DECL E6POS XP241={X 672,Y -551,Z 95,A 0,B 0,C 180,S 6,T 16,E1 0.0,E2 0.0,E3 0.0,E4 0.0,E5 0.0,E6 0.0}
DECL FDAT FP241={TOOL_NO 4,BASE_NO 0,IPO_FRAME #BASE,POINT2[] " "}
DECL LDAT LCPDAT241={VEL 1,ACC 50.000,APO_DIST 500.000,APO_FAC 50.0000,AXIS_VEL 50.000,AXIS_ACC 50.000,ORI_TYP #VAR,CIRC_TYP #BASE,JERK_FAC 50.0000,GEAR_JERK 100.000,EXAX_IGN 0}

DECL E6POS XP242={X 672,Y -601,Z 95,A 0,B 0,C 180,S 6,T 16,E1 0.0,E2 0.0,E3 0.0,E4 0.0,E5 0.0,E6 0.0}
DECL FDAT FP242={TOOL_NO 4,BASE_NO 0,IPO_FRAME #BASE,POINT2[] " "}
DECL LDAT LCPDAT242={VEL 1,ACC 50.000,APO_DIST 500.000,APO_FAC 50.0000,AXIS_VEL 50.000,AXIS_ACC 50.000,ORI_TYP #VAR,CIRC_TYP #BASE,JERK_FAC 50.0000,GEAR_JERK 100.000,EXAX_IGN 0}

DECL E6POS XP243={X 672,Y -651,Z 95,A 0,B 0,C 180,S 6,T 16,E1 0.0,E2 0.0,E3 0.0,E4 0.0,E5 0.0,E6 0.0}
DECL FDAT FP243={TOOL_NO 4,BASE_NO 0,IPO_FRAME #BASE,POINT2[] " "}
DECL LDAT LCPDAT243={VEL 1,ACC 50.000,APO_DIST 500.000,APO_FAC 50.0000,AXIS_VEL 50.000,AXIS_ACC 50.000,ORI_TYP #VAR,CIRC_TYP #BASE,JERK_FAC 50.0000,GEAR_JERK 100.000,EXAX_IGN 0}

DECL E6POS XP244={X 672,Y -651,Z 145,A 0,B 0,C 180,S 6,T 16,E1 0.0,E2 0.0,E3 0.0,E4 0.0,E5 0.0,E6 0.0}
DECL FDAT FP244={TOOL_NO 4,BASE_NO 0,IPO_FRAME #BASE,POINT2[] " "}
DECL LDAT LCPDAT244={VEL 1,ACC 50.000,APO_DIST 500.000,APO_FAC 50.0000,AXIS_VEL 50.000,AXIS_ACC 50.000,ORI_TYP #VAR,CIRC_TYP #BASE,JERK_FAC 50.0000,GEAR_JERK 100.000,EXAX_IGN 0}

DECL E6POS XP245={X 672,Y -601,Z 145,A 0,B 0,C 180,S 6,T 16,E1 0.0,E2 0.0,E3 0.0,E4 0.0,E5 0.0,E6 0.0}
DECL FDAT FP245={TOOL_NO 4,BASE_NO 0,IPO_FRAME #BASE,POINT2[] " "}
DECL LDAT LCPDAT245={VEL 1,ACC 50.000,APO_DIST 500.000,APO_FAC 50.0000,AXIS_VEL 50.000,AXIS_ACC 50.000,ORI_TYP #VAR,CIRC_TYP #BASE,JERK_FAC 50.0000,GEAR_JERK 100.000,EXAX_IGN 0}

DECL E6POS XP246={X 672,Y -551,Z 145,A 0,B 0,C 180,S 6,T 16,E1 0.0,E2 0.0,E3 0.0,E4 0.0,E5 0.0,E6 0.0}
DECL FDAT FP246={TOOL_NO 4,BASE_NO 0,IPO_FRAME #BASE,POINT2[] " "}
DECL LDAT LCPDAT246={VEL 1,ACC 50.000,APO_DIST 500.000,APO_FAC 50.0000,AXIS_VEL 50.000,AXIS_ACC 50.000,ORI_TYP #VAR,CIRC_TYP #BASE,JERK_FAC 50.0000,GEAR_JERK 100.000,EXAX_IGN 0}

DECL E6POS XP247={X 672,Y -501,Z 145,A 0,B 0,C 180,S 6,T 16,E1 0.0,E2 0.0,E3 0.0,E4 0.0,E5 0.0,E6 0.0}
DECL FDAT FP247={TOOL_NO 4,BASE_NO 0,IPO_FRAME #BASE,POINT2[] " "}
DECL LDAT LCPDAT247={VEL 1,ACC 50.000,APO_DIST 500.000,APO_FAC 50.0000,AXIS_VEL 50.000,AXIS_ACC 50.000,ORI_TYP #VAR,CIRC_TYP #BASE,JERK_FAC 50.0000,GEAR_JERK 100.000,EXAX_IGN 0}

DECL E6POS XP248={X 672,Y -451,Z 145,A 0,B 0,C 180,S 6,T 16,E1 0.0,E2 0.0,E3 0.0,E4 0.0,E5 0.0,E6 0.0}
DECL FDAT FP248={TOOL_NO 4,BASE_NO 0,IPO_FRAME #BASE,POINT2[] " "}
DECL LDAT LCPDAT248={VEL 1,ACC 50.000,APO_DIST 500.000,APO_FAC 50.0000,AXIS_VEL 50.000,AXIS_ACC 50.000,ORI_TYP #VAR,CIRC_TYP #BASE,JERK_FAC 50.0000,GEAR_JERK 100.000,EXAX_IGN 0}

DECL E6POS XP249={X 672,Y -401,Z 145,A 0,B 0,C 180,S 6,T 16,E1 0.0,E2 0.0,E3 0.0,E4 0.0,E5 0.0,E6 0.0}
DECL FDAT FP249={TOOL_NO 4,BASE_NO 0,IPO_FRAME #BASE,POINT2[] " "}
DECL LDAT LCPDAT249={VEL 1,ACC 50.000,APO_DIST 500.000,APO_FAC 50.0000,AXIS_VEL 50.000,AXIS_ACC 50.000,ORI_TYP #VAR,CIRC_TYP #BASE,JERK_FAC 50.0000,GEAR_JERK 100.000,EXAX_IGN 0}

DECL E6POS XP250={X 672,Y -351,Z 145,A 0,B 0,C 180,S 6,T 16,E1 0.0,E2 0.0,E3 0.0,E4 0.0,E5 0.0,E6 0.0}
DECL FDAT FP250={TOOL_NO 4,BASE_NO 0,IPO_FRAME #BASE,POINT2[] " "}
DECL LDAT LCPDAT250={VEL 1,ACC 50.000,APO_DIST 500.000,APO_FAC 50.0000,AXIS_VEL 50.000,AXIS_ACC 50.000,ORI_TYP #VAR,CIRC_TYP #BASE,JERK_FAC 50.0000,GEAR_JERK 100.000,EXAX_IGN 0}

DECL E6POS XP251={X 672,Y -301,Z 145,A 0,B 0,C 180,S 6,T 16,E1 0.0,E2 0.0,E3 0.0,E4 0.0,E5 0.0,E6 0.0}
DECL FDAT FP251={TOOL_NO 4,BASE_NO 0,IPO_FRAME #BASE,POINT2[] " "}
DECL LDAT LCPDAT251={VEL 1,ACC 50.000,APO_DIST 500.000,APO_FAC 50.0000,AXIS_VEL 50.000,AXIS_ACC 50.000,ORI_TYP #VAR,CIRC_TYP #BASE,JERK_FAC 50.0000,GEAR_JERK 100.000,EXAX_IGN 0}

DECL E6POS XP252={X 672,Y -251,Z 145,A 0,B 0,C 180,S 6,T 16,E1 0.0,E2 0.0,E3 0.0,E4 0.0,E5 0.0,E6 0.0}
DECL FDAT FP252={TOOL_NO 4,BASE_NO 0,IPO_FRAME #BASE,POINT2[] " "}
DECL LDAT LCPDAT252={VEL 1,ACC 50.000,APO_DIST 500.000,APO_FAC 50.0000,AXIS_VEL 50.000,AXIS_ACC 50.000,ORI_TYP #VAR,CIRC_TYP #BASE,JERK_FAC 50.0000,GEAR_JERK 100.000,EXAX_IGN 0}

DECL E6POS XP253={X 672,Y -201,Z 145,A 0,B 0,C 180,S 6,T 16,E1 0.0,E2 0.0,E3 0.0,E4 0.0,E5 0.0,E6 0.0}
DECL FDAT FP253={TOOL_NO 4,BASE_NO 0,IPO_FRAME #BASE,POINT2[] " "}
DECL LDAT LCPDAT253={VEL 1,ACC 50.000,APO_DIST 500.000,APO_FAC 50.0000,AXIS_VEL 50.000,AXIS_ACC 50.000,ORI_TYP #VAR,CIRC_TYP #BASE,JERK_FAC 50.0000,GEAR_JERK 100.000,EXAX_IGN 0}

DECL E6POS XP254={X 672,Y -151,Z 145,A 0,B 0,C 180,S 6,T 16,E1 0.0,E2 0.0,E3 0.0,E4 0.0,E5 0.0,E6 0.0}
DECL FDAT FP254={TOOL_NO 4,BASE_NO 0,IPO_FRAME #BASE,POINT2[] " "}
DECL LDAT LCPDAT254={VEL 1,ACC 50.000,APO_DIST 500.000,APO_FAC 50.0000,AXIS_VEL 50.000,AXIS_ACC 50.000,ORI_TYP #VAR,CIRC_TYP #BASE,JERK_FAC 50.0000,GEAR_JERK 100.000,EXAX_IGN 0}

DECL E6POS XP255={X 672,Y -101,Z 145,A 0,B 0,C 180,S 6,T 16,E1 0.0,E2 0.0,E3 0.0,E4 0.0,E5 0.0,E6 0.0}
DECL FDAT FP255={TOOL_NO 4,BASE_NO 0,IPO_FRAME #BASE,POINT2[] " "}
DECL LDAT LCPDAT255={VEL 1,ACC 50.000,APO_DIST 500.000,APO_FAC 50.0000,AXIS_VEL 50.000,AXIS_ACC 50.000,ORI_TYP #VAR,CIRC_TYP #BASE,JERK_FAC 50.0000,GEAR_JERK 100.000,EXAX_IGN 0}

DECL E6POS XP256={X 672,Y -51,Z 145,A 0,B 0,C 180,S 6,T 16,E1 0.0,E2 0.0,E3 0.0,E4 0.0,E5 0.0,E6 0.0}
DECL FDAT FP256={TOOL_NO 4,BASE_NO 0,IPO_FRAME #BASE,POINT2[] " "}
DECL LDAT LCPDAT256={VEL 1,ACC 50.000,APO_DIST 500.000,APO_FAC 50.0000,AXIS_VEL 50.000,AXIS_ACC 50.000,ORI_TYP #VAR,CIRC_TYP #BASE,JERK_FAC 50.0000,GEAR_JERK 100.000,EXAX_IGN 0}

DECL E6POS XP257={X 672,Y -1,Z 145,A 0,B 0,C 180,S 6,T 16,E1 0.0,E2 0.0,E3 0.0,E4 0.0,E5 0.0,E6 0.0}
DECL FDAT FP257={TOOL_NO 4,BASE_NO 0,IPO_FRAME #BASE,POINT2[] " "}
DECL LDAT LCPDAT257={VEL 1,ACC 50.000,APO_DIST 500.000,APO_FAC 50.0000,AXIS_VEL 50.000,AXIS_ACC 50.000,ORI_TYP #VAR,CIRC_TYP #BASE,JERK_FAC 50.0000,GEAR_JERK 100.000,EXAX_IGN 0}

DECL E6POS XP258={X 672,Y 49,Z 145,A 0,B 0,C 180,S 6,T 16,E1 0.0,E2 0.0,E3 0.0,E4 0.0,E5 0.0,E6 0.0}
DECL FDAT FP258={TOOL_NO 4,BASE_NO 0,IPO_FRAME #BASE,POINT2[] " "}
DECL LDAT LCPDAT258={VEL 1,ACC 50.000,APO_DIST 500.000,APO_FAC 50.0000,AXIS_VEL 50.000,AXIS_ACC 50.000,ORI_TYP #VAR,CIRC_TYP #BASE,JERK_FAC 50.0000,GEAR_JERK 100.000,EXAX_IGN 0}

DECL E6POS XP259={X 672,Y 99,Z 145,A 0,B 0,C 180,S 6,T 16,E1 0.0,E2 0.0,E3 0.0,E4 0.0,E5 0.0,E6 0.0}
DECL FDAT FP259={TOOL_NO 4,BASE_NO 0,IPO_FRAME #BASE,POINT2[] " "}
DECL LDAT LCPDAT259={VEL 1,ACC 50.000,APO_DIST 500.000,APO_FAC 50.0000,AXIS_VEL 50.000,AXIS_ACC 50.000,ORI_TYP #VAR,CIRC_TYP #BASE,JERK_FAC 50.0000,GEAR_JERK 100.000,EXAX_IGN 0}

DECL E6POS XP260={X 672,Y 149,Z 145,A 0,B 0,C 180,S 6,T 16,E1 0.0,E2 0.0,E3 0.0,E4 0.0,E5 0.0,E6 0.0}
DECL FDAT FP260={TOOL_NO 4,BASE_NO 0,IPO_FRAME #BASE,POINT2[] " "}
DECL LDAT LCPDAT260={VEL 1,ACC 50.000,APO_DIST 500.000,APO_FAC 50.0000,AXIS_VEL 50.000,AXIS_ACC 50.000,ORI_TYP #VAR,CIRC_TYP #BASE,JERK_FAC 50.0000,GEAR_JERK 100.000,EXAX_IGN 0}

DECL E6POS XP261={X 672,Y 199,Z 145,A 0,B 0,C 180,S 6,T 16,E1 0.0,E2 0.0,E3 0.0,E4 0.0,E5 0.0,E6 0.0}
DECL FDAT FP261={TOOL_NO 4,BASE_NO 0,IPO_FRAME #BASE,POINT2[] " "}
DECL LDAT LCPDAT261={VEL 1,ACC 50.000,APO_DIST 500.000,APO_FAC 50.0000,AXIS_VEL 50.000,AXIS_ACC 50.000,ORI_TYP #VAR,CIRC_TYP #BASE,JERK_FAC 50.0000,GEAR_JERK 100.000,EXAX_IGN 0}

DECL E6POS XP262={X 672,Y 249,Z 145,A 0,B 0,C 180,S 6,T 16,E1 0.0,E2 0.0,E3 0.0,E4 0.0,E5 0.0,E6 0.0}
DECL FDAT FP262={TOOL_NO 4,BASE_NO 0,IPO_FRAME #BASE,POINT2[] " "}
DECL LDAT LCPDAT262={VEL 1,ACC 50.000,APO_DIST 500.000,APO_FAC 50.0000,AXIS_VEL 50.000,AXIS_ACC 50.000,ORI_TYP #VAR,CIRC_TYP #BASE,JERK_FAC 50.0000,GEAR_JERK 100.000,EXAX_IGN 0}

DECL E6POS XP263={X 672,Y 299,Z 145,A 0,B 0,C 180,S 6,T 16,E1 0.0,E2 0.0,E3 0.0,E4 0.0,E5 0.0,E6 0.0}
DECL FDAT FP263={TOOL_NO 4,BASE_NO 0,IPO_FRAME #BASE,POINT2[] " "}
DECL LDAT LCPDAT263={VEL 1,ACC 50.000,APO_DIST 500.000,APO_FAC 50.0000,AXIS_VEL 50.000,AXIS_ACC 50.000,ORI_TYP #VAR,CIRC_TYP #BASE,JERK_FAC 50.0000,GEAR_JERK 100.000,EXAX_IGN 0}

DECL E6POS XP264={X 672,Y 349,Z 145,A 0,B 0,C 180,S 6,T 16,E1 0.0,E2 0.0,E3 0.0,E4 0.0,E5 0.0,E6 0.0}
DECL FDAT FP264={TOOL_NO 4,BASE_NO 0,IPO_FRAME #BASE,POINT2[] " "}
DECL LDAT LCPDAT264={VEL 1,ACC 50.000,APO_DIST 500.000,APO_FAC 50.0000,AXIS_VEL 50.000,AXIS_ACC 50.000,ORI_TYP #VAR,CIRC_TYP #BASE,JERK_FAC 50.0000,GEAR_JERK 100.000,EXAX_IGN 0}

DECL E6POS XP265={X 672,Y 399,Z 145,A 0,B 0,C 180,S 6,T 16,E1 0.0,E2 0.0,E3 0.0,E4 0.0,E5 0.0,E6 0.0}
DECL FDAT FP265={TOOL_NO 4,BASE_NO 0,IPO_FRAME #BASE,POINT2[] " "}
DECL LDAT LCPDAT265={VEL 1,ACC 50.000,APO_DIST 500.000,APO_FAC 50.0000,AXIS_VEL 50.000,AXIS_ACC 50.000,ORI_TYP #VAR,CIRC_TYP #BASE,JERK_FAC 50.0000,GEAR_JERK 100.000,EXAX_IGN 0}

DECL E6POS XP266={X 672,Y 449,Z 145,A 0,B 0,C 180,S 6,T 16,E1 0.0,E2 0.0,E3 0.0,E4 0.0,E5 0.0,E6 0.0}
DECL FDAT FP266={TOOL_NO 4,BASE_NO 0,IPO_FRAME #BASE,POINT2[] " "}
DECL LDAT LCPDAT266={VEL 1,ACC 50.000,APO_DIST 500.000,APO_FAC 50.0000,AXIS_VEL 50.000,AXIS_ACC 50.000,ORI_TYP #VAR,CIRC_TYP #BASE,JERK_FAC 50.0000,GEAR_JERK 100.000,EXAX_IGN 0}

DECL E6POS XP267={X 672,Y 499,Z 145,A 0,B 0,C 180,S 6,T 16,E1 0.0,E2 0.0,E3 0.0,E4 0.0,E5 0.0,E6 0.0}
DECL FDAT FP267={TOOL_NO 4,BASE_NO 0,IPO_FRAME #BASE,POINT2[] " "}
DECL LDAT LCPDAT267={VEL 1,ACC 50.000,APO_DIST 500.000,APO_FAC 50.0000,AXIS_VEL 50.000,AXIS_ACC 50.000,ORI_TYP #VAR,CIRC_TYP #BASE,JERK_FAC 50.0000,GEAR_JERK 100.000,EXAX_IGN 0}

DECL E6POS XP268={X 672,Y 499,Z 195,A 0,B 0,C 180,S 6,T 16,E1 0.0,E2 0.0,E3 0.0,E4 0.0,E5 0.0,E6 0.0}
DECL FDAT FP268={TOOL_NO 4,BASE_NO 0,IPO_FRAME #BASE,POINT2[] " "}
DECL LDAT LCPDAT268={VEL 1,ACC 50.000,APO_DIST 500.000,APO_FAC 50.0000,AXIS_VEL 50.000,AXIS_ACC 50.000,ORI_TYP #VAR,CIRC_TYP #BASE,JERK_FAC 50.0000,GEAR_JERK 100.000,EXAX_IGN 0}

DECL E6POS XP269={X 672,Y 449,Z 195,A 0,B 0,C 180,S 6,T 16,E1 0.0,E2 0.0,E3 0.0,E4 0.0,E5 0.0,E6 0.0}
DECL FDAT FP269={TOOL_NO 4,BASE_NO 0,IPO_FRAME #BASE,POINT2[] " "}
DECL LDAT LCPDAT269={VEL 1,ACC 50.000,APO_DIST 500.000,APO_FAC 50.0000,AXIS_VEL 50.000,AXIS_ACC 50.000,ORI_TYP #VAR,CIRC_TYP #BASE,JERK_FAC 50.0000,GEAR_JERK 100.000,EXAX_IGN 0}

DECL E6POS XP270={X 672,Y 399,Z 195,A 0,B 0,C 180,S 6,T 16,E1 0.0,E2 0.0,E3 0.0,E4 0.0,E5 0.0,E6 0.0}
DECL FDAT FP270={TOOL_NO 4,BASE_NO 0,IPO_FRAME #BASE,POINT2[] " "}
DECL LDAT LCPDAT270={VEL 1,ACC 50.000,APO_DIST 500.000,APO_FAC 50.0000,AXIS_VEL 50.000,AXIS_ACC 50.000,ORI_TYP #VAR,CIRC_TYP #BASE,JERK_FAC 50.0000,GEAR_JERK 100.000,EXAX_IGN 0}

DECL E6POS XP271={X 672,Y 349,Z 195,A 0,B 0,C 180,S 6,T 16,E1 0.0,E2 0.0,E3 0.0,E4 0.0,E5 0.0,E6 0.0}
DECL FDAT FP271={TOOL_NO 4,BASE_NO 0,IPO_FRAME #BASE,POINT2[] " "}
DECL LDAT LCPDAT271={VEL 1,ACC 50.000,APO_DIST 500.000,APO_FAC 50.0000,AXIS_VEL 50.000,AXIS_ACC 50.000,ORI_TYP #VAR,CIRC_TYP #BASE,JERK_FAC 50.0000,GEAR_JERK 100.000,EXAX_IGN 0}

DECL E6POS XP272={X 672,Y 299,Z 195,A 0,B 0,C 180,S 6,T 16,E1 0.0,E2 0.0,E3 0.0,E4 0.0,E5 0.0,E6 0.0}
DECL FDAT FP272={TOOL_NO 4,BASE_NO 0,IPO_FRAME #BASE,POINT2[] " "}
DECL LDAT LCPDAT272={VEL 1,ACC 50.000,APO_DIST 500.000,APO_FAC 50.0000,AXIS_VEL 50.000,AXIS_ACC 50.000,ORI_TYP #VAR,CIRC_TYP #BASE,JERK_FAC 50.0000,GEAR_JERK 100.000,EXAX_IGN 0}

DECL E6POS XP273={X 672,Y 249,Z 195,A 0,B 0,C 180,S 6,T 16,E1 0.0,E2 0.0,E3 0.0,E4 0.0,E5 0.0,E6 0.0}
DECL FDAT FP273={TOOL_NO 4,BASE_NO 0,IPO_FRAME #BASE,POINT2[] " "}
DECL LDAT LCPDAT273={VEL 1,ACC 50.000,APO_DIST 500.000,APO_FAC 50.0000,AXIS_VEL 50.000,AXIS_ACC 50.000,ORI_TYP #VAR,CIRC_TYP #BASE,JERK_FAC 50.0000,GEAR_JERK 100.000,EXAX_IGN 0}

DECL E6POS XP274={X 672,Y 199,Z 195,A 0,B 0,C 180,S 6,T 16,E1 0.0,E2 0.0,E3 0.0,E4 0.0,E5 0.0,E6 0.0}
DECL FDAT FP274={TOOL_NO 4,BASE_NO 0,IPO_FRAME #BASE,POINT2[] " "}
DECL LDAT LCPDAT274={VEL 1,ACC 50.000,APO_DIST 500.000,APO_FAC 50.0000,AXIS_VEL 50.000,AXIS_ACC 50.000,ORI_TYP #VAR,CIRC_TYP #BASE,JERK_FAC 50.0000,GEAR_JERK 100.000,EXAX_IGN 0}

DECL E6POS XP275={X 672,Y 149,Z 195,A 0,B 0,C 180,S 6,T 16,E1 0.0,E2 0.0,E3 0.0,E4 0.0,E5 0.0,E6 0.0}
DECL FDAT FP275={TOOL_NO 4,BASE_NO 0,IPO_FRAME #BASE,POINT2[] " "}
DECL LDAT LCPDAT275={VEL 1,ACC 50.000,APO_DIST 500.000,APO_FAC 50.0000,AXIS_VEL 50.000,AXIS_ACC 50.000,ORI_TYP #VAR,CIRC_TYP #BASE,JERK_FAC 50.0000,GEAR_JERK 100.000,EXAX_IGN 0}

DECL E6POS XP276={X 672,Y 99,Z 195,A 0,B 0,C 180,S 6,T 16,E1 0.0,E2 0.0,E3 0.0,E4 0.0,E5 0.0,E6 0.0}
DECL FDAT FP276={TOOL_NO 4,BASE_NO 0,IPO_FRAME #BASE,POINT2[] " "}
DECL LDAT LCPDAT276={VEL 1,ACC 50.000,APO_DIST 500.000,APO_FAC 50.0000,AXIS_VEL 50.000,AXIS_ACC 50.000,ORI_TYP #VAR,CIRC_TYP #BASE,JERK_FAC 50.0000,GEAR_JERK 100.000,EXAX_IGN 0}

DECL E6POS XP277={X 672,Y 49,Z 195,A 0,B 0,C 180,S 6,T 16,E1 0.0,E2 0.0,E3 0.0,E4 0.0,E5 0.0,E6 0.0}
DECL FDAT FP277={TOOL_NO 4,BASE_NO 0,IPO_FRAME #BASE,POINT2[] " "}
DECL LDAT LCPDAT277={VEL 1,ACC 50.000,APO_DIST 500.000,APO_FAC 50.0000,AXIS_VEL 50.000,AXIS_ACC 50.000,ORI_TYP #VAR,CIRC_TYP #BASE,JERK_FAC 50.0000,GEAR_JERK 100.000,EXAX_IGN 0}

DECL E6POS XP278={X 672,Y -1,Z 195,A 0,B 0,C 180,S 6,T 16,E1 0.0,E2 0.0,E3 0.0,E4 0.0,E5 0.0,E6 0.0}
DECL FDAT FP278={TOOL_NO 4,BASE_NO 0,IPO_FRAME #BASE,POINT2[] " "}
DECL LDAT LCPDAT278={VEL 1,ACC 50.000,APO_DIST 500.000,APO_FAC 50.0000,AXIS_VEL 50.000,AXIS_ACC 50.000,ORI_TYP #VAR,CIRC_TYP #BASE,JERK_FAC 50.0000,GEAR_JERK 100.000,EXAX_IGN 0}

DECL E6POS XP279={X 672,Y -51,Z 195,A 0,B 0,C 180,S 6,T 16,E1 0.0,E2 0.0,E3 0.0,E4 0.0,E5 0.0,E6 0.0}
DECL FDAT FP279={TOOL_NO 4,BASE_NO 0,IPO_FRAME #BASE,POINT2[] " "}
DECL LDAT LCPDAT279={VEL 1,ACC 50.000,APO_DIST 500.000,APO_FAC 50.0000,AXIS_VEL 50.000,AXIS_ACC 50.000,ORI_TYP #VAR,CIRC_TYP #BASE,JERK_FAC 50.0000,GEAR_JERK 100.000,EXAX_IGN 0}

DECL E6POS XP280={X 672,Y -101,Z 195,A 0,B 0,C 180,S 6,T 16,E1 0.0,E2 0.0,E3 0.0,E4 0.0,E5 0.0,E6 0.0}
DECL FDAT FP280={TOOL_NO 4,BASE_NO 0,IPO_FRAME #BASE,POINT2[] " "}
DECL LDAT LCPDAT280={VEL 1,ACC 50.000,APO_DIST 500.000,APO_FAC 50.0000,AXIS_VEL 50.000,AXIS_ACC 50.000,ORI_TYP #VAR,CIRC_TYP #BASE,JERK_FAC 50.0000,GEAR_JERK 100.000,EXAX_IGN 0}

DECL E6POS XP281={X 672,Y -151,Z 195,A 0,B 0,C 180,S 6,T 16,E1 0.0,E2 0.0,E3 0.0,E4 0.0,E5 0.0,E6 0.0}
DECL FDAT FP281={TOOL_NO 4,BASE_NO 0,IPO_FRAME #BASE,POINT2[] " "}
DECL LDAT LCPDAT281={VEL 1,ACC 50.000,APO_DIST 500.000,APO_FAC 50.0000,AXIS_VEL 50.000,AXIS_ACC 50.000,ORI_TYP #VAR,CIRC_TYP #BASE,JERK_FAC 50.0000,GEAR_JERK 100.000,EXAX_IGN 0}

DECL E6POS XP282={X 672,Y -201,Z 195,A 0,B 0,C 180,S 6,T 16,E1 0.0,E2 0.0,E3 0.0,E4 0.0,E5 0.0,E6 0.0}
DECL FDAT FP282={TOOL_NO 4,BASE_NO 0,IPO_FRAME #BASE,POINT2[] " "}
DECL LDAT LCPDAT282={VEL 1,ACC 50.000,APO_DIST 500.000,APO_FAC 50.0000,AXIS_VEL 50.000,AXIS_ACC 50.000,ORI_TYP #VAR,CIRC_TYP #BASE,JERK_FAC 50.0000,GEAR_JERK 100.000,EXAX_IGN 0}

DECL E6POS XP283={X 672,Y -251,Z 195,A 0,B 0,C 180,S 6,T 16,E1 0.0,E2 0.0,E3 0.0,E4 0.0,E5 0.0,E6 0.0}
DECL FDAT FP283={TOOL_NO 4,BASE_NO 0,IPO_FRAME #BASE,POINT2[] " "}
DECL LDAT LCPDAT283={VEL 1,ACC 50.000,APO_DIST 500.000,APO_FAC 50.0000,AXIS_VEL 50.000,AXIS_ACC 50.000,ORI_TYP #VAR,CIRC_TYP #BASE,JERK_FAC 50.0000,GEAR_JERK 100.000,EXAX_IGN 0}

DECL E6POS XP284={X 672,Y -301,Z 195,A 0,B 0,C 180,S 6,T 16,E1 0.0,E2 0.0,E3 0.0,E4 0.0,E5 0.0,E6 0.0}
DECL FDAT FP284={TOOL_NO 4,BASE_NO 0,IPO_FRAME #BASE,POINT2[] " "}
DECL LDAT LCPDAT284={VEL 1,ACC 50.000,APO_DIST 500.000,APO_FAC 50.0000,AXIS_VEL 50.000,AXIS_ACC 50.000,ORI_TYP #VAR,CIRC_TYP #BASE,JERK_FAC 50.0000,GEAR_JERK 100.000,EXAX_IGN 0}

DECL E6POS XP285={X 672,Y -351,Z 195,A 0,B 0,C 180,S 6,T 16,E1 0.0,E2 0.0,E3 0.0,E4 0.0,E5 0.0,E6 0.0}
DECL FDAT FP285={TOOL_NO 4,BASE_NO 0,IPO_FRAME #BASE,POINT2[] " "}
DECL LDAT LCPDAT285={VEL 1,ACC 50.000,APO_DIST 500.000,APO_FAC 50.0000,AXIS_VEL 50.000,AXIS_ACC 50.000,ORI_TYP #VAR,CIRC_TYP #BASE,JERK_FAC 50.0000,GEAR_JERK 100.000,EXAX_IGN 0}

DECL E6POS XP286={X 672,Y -401,Z 195,A 0,B 0,C 180,S 6,T 16,E1 0.0,E2 0.0,E3 0.0,E4 0.0,E5 0.0,E6 0.0}
DECL FDAT FP286={TOOL_NO 4,BASE_NO 0,IPO_FRAME #BASE,POINT2[] " "}
DECL LDAT LCPDAT286={VEL 1,ACC 50.000,APO_DIST 500.000,APO_FAC 50.0000,AXIS_VEL 50.000,AXIS_ACC 50.000,ORI_TYP #VAR,CIRC_TYP #BASE,JERK_FAC 50.0000,GEAR_JERK 100.000,EXAX_IGN 0}

DECL E6POS XP287={X 672,Y -451,Z 195,A 0,B 0,C 180,S 6,T 16,E1 0.0,E2 0.0,E3 0.0,E4 0.0,E5 0.0,E6 0.0}
DECL FDAT FP287={TOOL_NO 4,BASE_NO 0,IPO_FRAME #BASE,POINT2[] " "}
DECL LDAT LCPDAT287={VEL 1,ACC 50.000,APO_DIST 500.000,APO_FAC 50.0000,AXIS_VEL 50.000,AXIS_ACC 50.000,ORI_TYP #VAR,CIRC_TYP #BASE,JERK_FAC 50.0000,GEAR_JERK 100.000,EXAX_IGN 0}

DECL E6POS XP288={X 672,Y -501,Z 195,A 0,B 0,C 180,S 6,T 16,E1 0.0,E2 0.0,E3 0.0,E4 0.0,E5 0.0,E6 0.0}
DECL FDAT FP288={TOOL_NO 4,BASE_NO 0,IPO_FRAME #BASE,POINT2[] " "}
DECL LDAT LCPDAT288={VEL 1,ACC 50.000,APO_DIST 500.000,APO_FAC 50.0000,AXIS_VEL 50.000,AXIS_ACC 50.000,ORI_TYP #VAR,CIRC_TYP #BASE,JERK_FAC 50.0000,GEAR_JERK 100.000,EXAX_IGN 0}

DECL E6POS XP289={X 672,Y -551,Z 195,A 0,B 0,C 180,S 6,T 16,E1 0.0,E2 0.0,E3 0.0,E4 0.0,E5 0.0,E6 0.0}
DECL FDAT FP289={TOOL_NO 4,BASE_NO 0,IPO_FRAME #BASE,POINT2[] " "}
DECL LDAT LCPDAT289={VEL 1,ACC 50.000,APO_DIST 500.000,APO_FAC 50.0000,AXIS_VEL 50.000,AXIS_ACC 50.000,ORI_TYP #VAR,CIRC_TYP #BASE,JERK_FAC 50.0000,GEAR_JERK 100.000,EXAX_IGN 0}

DECL E6POS XP290={X 672,Y -601,Z 195,A 0,B 0,C 180,S 6,T 16,E1 0.0,E2 0.0,E3 0.0,E4 0.0,E5 0.0,E6 0.0}
DECL FDAT FP290={TOOL_NO 4,BASE_NO 0,IPO_FRAME #BASE,POINT2[] " "}
DECL LDAT LCPDAT290={VEL 1,ACC 50.000,APO_DIST 500.000,APO_FAC 50.0000,AXIS_VEL 50.000,AXIS_ACC 50.000,ORI_TYP #VAR,CIRC_TYP #BASE,JERK_FAC 50.0000,GEAR_JERK 100.000,EXAX_IGN 0}

DECL E6POS XP291={X 672,Y -651,Z 195,A 0,B 0,C 180,S 6,T 16,E1 0.0,E2 0.0,E3 0.0,E4 0.0,E5 0.0,E6 0.0}
DECL FDAT FP291={TOOL_NO 4,BASE_NO 0,IPO_FRAME #BASE,POINT2[] " "}
DECL LDAT LCPDAT291={VEL 1,ACC 50.000,APO_DIST 500.000,APO_FAC 50.0000,AXIS_VEL 50.000,AXIS_ACC 50.000,ORI_TYP #VAR,CIRC_TYP #BASE,JERK_FAC 50.0000,GEAR_JERK 100.000,EXAX_IGN 0}

DECL E6POS XP292={X 672,Y -651,Z 245,A 0,B 0,C 180,S 6,T 16,E1 0.0,E2 0.0,E3 0.0,E4 0.0,E5 0.0,E6 0.0}
DECL FDAT FP292={TOOL_NO 4,BASE_NO 0,IPO_FRAME #BASE,POINT2[] " "}
DECL LDAT LCPDAT292={VEL 1,ACC 50.000,APO_DIST 500.000,APO_FAC 50.0000,AXIS_VEL 50.000,AXIS_ACC 50.000,ORI_TYP #VAR,CIRC_TYP #BASE,JERK_FAC 50.0000,GEAR_JERK 100.000,EXAX_IGN 0}

DECL E6POS XP293={X 672,Y -601,Z 245,A 0,B 0,C 180,S 6,T 16,E1 0.0,E2 0.0,E3 0.0,E4 0.0,E5 0.0,E6 0.0}
DECL FDAT FP293={TOOL_NO 4,BASE_NO 0,IPO_FRAME #BASE,POINT2[] " "}
DECL LDAT LCPDAT293={VEL 1,ACC 50.000,APO_DIST 500.000,APO_FAC 50.0000,AXIS_VEL 50.000,AXIS_ACC 50.000,ORI_TYP #VAR,CIRC_TYP #BASE,JERK_FAC 50.0000,GEAR_JERK 100.000,EXAX_IGN 0}

DECL E6POS XP294={X 672,Y -551,Z 245,A 0,B 0,C 180,S 6,T 16,E1 0.0,E2 0.0,E3 0.0,E4 0.0,E5 0.0,E6 0.0}
DECL FDAT FP294={TOOL_NO 4,BASE_NO 0,IPO_FRAME #BASE,POINT2[] " "}
DECL LDAT LCPDAT294={VEL 1,ACC 50.000,APO_DIST 500.000,APO_FAC 50.0000,AXIS_VEL 50.000,AXIS_ACC 50.000,ORI_TYP #VAR,CIRC_TYP #BASE,JERK_FAC 50.0000,GEAR_JERK 100.000,EXAX_IGN 0}

DECL E6POS XP295={X 672,Y -501,Z 245,A 0,B 0,C 180,S 6,T 16,E1 0.0,E2 0.0,E3 0.0,E4 0.0,E5 0.0,E6 0.0}
DECL FDAT FP295={TOOL_NO 4,BASE_NO 0,IPO_FRAME #BASE,POINT2[] " "}
DECL LDAT LCPDAT295={VEL 1,ACC 50.000,APO_DIST 500.000,APO_FAC 50.0000,AXIS_VEL 50.000,AXIS_ACC 50.000,ORI_TYP #VAR,CIRC_TYP #BASE,JERK_FAC 50.0000,GEAR_JERK 100.000,EXAX_IGN 0}

DECL E6POS XP296={X 672,Y -451,Z 245,A 0,B 0,C 180,S 6,T 16,E1 0.0,E2 0.0,E3 0.0,E4 0.0,E5 0.0,E6 0.0}
DECL FDAT FP296={TOOL_NO 4,BASE_NO 0,IPO_FRAME #BASE,POINT2[] " "}
DECL LDAT LCPDAT296={VEL 1,ACC 50.000,APO_DIST 500.000,APO_FAC 50.0000,AXIS_VEL 50.000,AXIS_ACC 50.000,ORI_TYP #VAR,CIRC_TYP #BASE,JERK_FAC 50.0000,GEAR_JERK 100.000,EXAX_IGN 0}

DECL E6POS XP297={X 672,Y -401,Z 245,A 0,B 0,C 180,S 6,T 16,E1 0.0,E2 0.0,E3 0.0,E4 0.0,E5 0.0,E6 0.0}
DECL FDAT FP297={TOOL_NO 4,BASE_NO 0,IPO_FRAME #BASE,POINT2[] " "}
DECL LDAT LCPDAT297={VEL 1,ACC 50.000,APO_DIST 500.000,APO_FAC 50.0000,AXIS_VEL 50.000,AXIS_ACC 50.000,ORI_TYP #VAR,CIRC_TYP #BASE,JERK_FAC 50.0000,GEAR_JERK 100.000,EXAX_IGN 0}

DECL E6POS XP298={X 672,Y -351,Z 245,A 0,B 0,C 180,S 6,T 16,E1 0.0,E2 0.0,E3 0.0,E4 0.0,E5 0.0,E6 0.0}
DECL FDAT FP298={TOOL_NO 4,BASE_NO 0,IPO_FRAME #BASE,POINT2[] " "}
DECL LDAT LCPDAT298={VEL 1,ACC 50.000,APO_DIST 500.000,APO_FAC 50.0000,AXIS_VEL 50.000,AXIS_ACC 50.000,ORI_TYP #VAR,CIRC_TYP #BASE,JERK_FAC 50.0000,GEAR_JERK 100.000,EXAX_IGN 0}

DECL E6POS XP299={X 672,Y -301,Z 245,A 0,B 0,C 180,S 6,T 16,E1 0.0,E2 0.0,E3 0.0,E4 0.0,E5 0.0,E6 0.0}
DECL FDAT FP299={TOOL_NO 4,BASE_NO 0,IPO_FRAME #BASE,POINT2[] " "}
DECL LDAT LCPDAT299={VEL 1,ACC 50.000,APO_DIST 500.000,APO_FAC 50.0000,AXIS_VEL 50.000,AXIS_ACC 50.000,ORI_TYP #VAR,CIRC_TYP #BASE,JERK_FAC 50.0000,GEAR_JERK 100.000,EXAX_IGN 0}

DECL E6POS XP300={X 672,Y -251,Z 245,A 0,B 0,C 180,S 6,T 16,E1 0.0,E2 0.0,E3 0.0,E4 0.0,E5 0.0,E6 0.0}
DECL FDAT FP300={TOOL_NO 4,BASE_NO 0,IPO_FRAME #BASE,POINT2[] " "}
DECL LDAT LCPDAT300={VEL 1,ACC 50.000,APO_DIST 500.000,APO_FAC 50.0000,AXIS_VEL 50.000,AXIS_ACC 50.000,ORI_TYP #VAR,CIRC_TYP #BASE,JERK_FAC 50.0000,GEAR_JERK 100.000,EXAX_IGN 0}

DECL E6POS XP301={X 672,Y -201,Z 245,A 0,B 0,C 180,S 6,T 16,E1 0.0,E2 0.0,E3 0.0,E4 0.0,E5 0.0,E6 0.0}
DECL FDAT FP301={TOOL_NO 4,BASE_NO 0,IPO_FRAME #BASE,POINT2[] " "}
DECL LDAT LCPDAT301={VEL 1,ACC 50.000,APO_DIST 500.000,APO_FAC 50.0000,AXIS_VEL 50.000,AXIS_ACC 50.000,ORI_TYP #VAR,CIRC_TYP #BASE,JERK_FAC 50.0000,GEAR_JERK 100.000,EXAX_IGN 0}

DECL E6POS XP302={X 672,Y -151,Z 245,A 0,B 0,C 180,S 6,T 16,E1 0.0,E2 0.0,E3 0.0,E4 0.0,E5 0.0,E6 0.0}
DECL FDAT FP302={TOOL_NO 4,BASE_NO 0,IPO_FRAME #BASE,POINT2[] " "}
DECL LDAT LCPDAT302={VEL 1,ACC 50.000,APO_DIST 500.000,APO_FAC 50.0000,AXIS_VEL 50.000,AXIS_ACC 50.000,ORI_TYP #VAR,CIRC_TYP #BASE,JERK_FAC 50.0000,GEAR_JERK 100.000,EXAX_IGN 0}

DECL E6POS XP303={X 672,Y -101,Z 245,A 0,B 0,C 180,S 6,T 16,E1 0.0,E2 0.0,E3 0.0,E4 0.0,E5 0.0,E6 0.0}
DECL FDAT FP303={TOOL_NO 4,BASE_NO 0,IPO_FRAME #BASE,POINT2[] " "}
DECL LDAT LCPDAT303={VEL 1,ACC 50.000,APO_DIST 500.000,APO_FAC 50.0000,AXIS_VEL 50.000,AXIS_ACC 50.000,ORI_TYP #VAR,CIRC_TYP #BASE,JERK_FAC 50.0000,GEAR_JERK 100.000,EXAX_IGN 0}

DECL E6POS XP304={X 672,Y -51,Z 245,A 0,B 0,C 180,S 6,T 16,E1 0.0,E2 0.0,E3 0.0,E4 0.0,E5 0.0,E6 0.0}
DECL FDAT FP304={TOOL_NO 4,BASE_NO 0,IPO_FRAME #BASE,POINT2[] " "}
DECL LDAT LCPDAT304={VEL 1,ACC 50.000,APO_DIST 500.000,APO_FAC 50.0000,AXIS_VEL 50.000,AXIS_ACC 50.000,ORI_TYP #VAR,CIRC_TYP #BASE,JERK_FAC 50.0000,GEAR_JERK 100.000,EXAX_IGN 0}

DECL E6POS XP305={X 672,Y -1,Z 245,A 0,B 0,C 180,S 6,T 16,E1 0.0,E2 0.0,E3 0.0,E4 0.0,E5 0.0,E6 0.0}
DECL FDAT FP305={TOOL_NO 4,BASE_NO 0,IPO_FRAME #BASE,POINT2[] " "}
DECL LDAT LCPDAT305={VEL 1,ACC 50.000,APO_DIST 500.000,APO_FAC 50.0000,AXIS_VEL 50.000,AXIS_ACC 50.000,ORI_TYP #VAR,CIRC_TYP #BASE,JERK_FAC 50.0000,GEAR_JERK 100.000,EXAX_IGN 0}

DECL E6POS XP306={X 672,Y 49,Z 245,A 0,B 0,C 180,S 6,T 16,E1 0.0,E2 0.0,E3 0.0,E4 0.0,E5 0.0,E6 0.0}
DECL FDAT FP306={TOOL_NO 4,BASE_NO 0,IPO_FRAME #BASE,POINT2[] " "}
DECL LDAT LCPDAT306={VEL 1,ACC 50.000,APO_DIST 500.000,APO_FAC 50.0000,AXIS_VEL 50.000,AXIS_ACC 50.000,ORI_TYP #VAR,CIRC_TYP #BASE,JERK_FAC 50.0000,GEAR_JERK 100.000,EXAX_IGN 0}

DECL E6POS XP307={X 672,Y 99,Z 245,A 0,B 0,C 180,S 6,T 16,E1 0.0,E2 0.0,E3 0.0,E4 0.0,E5 0.0,E6 0.0}
DECL FDAT FP307={TOOL_NO 4,BASE_NO 0,IPO_FRAME #BASE,POINT2[] " "}
DECL LDAT LCPDAT307={VEL 1,ACC 50.000,APO_DIST 500.000,APO_FAC 50.0000,AXIS_VEL 50.000,AXIS_ACC 50.000,ORI_TYP #VAR,CIRC_TYP #BASE,JERK_FAC 50.0000,GEAR_JERK 100.000,EXAX_IGN 0}

DECL E6POS XP308={X 672,Y 149,Z 245,A 0,B 0,C 180,S 6,T 16,E1 0.0,E2 0.0,E3 0.0,E4 0.0,E5 0.0,E6 0.0}
DECL FDAT FP308={TOOL_NO 4,BASE_NO 0,IPO_FRAME #BASE,POINT2[] " "}
DECL LDAT LCPDAT308={VEL 1,ACC 50.000,APO_DIST 500.000,APO_FAC 50.0000,AXIS_VEL 50.000,AXIS_ACC 50.000,ORI_TYP #VAR,CIRC_TYP #BASE,JERK_FAC 50.0000,GEAR_JERK 100.000,EXAX_IGN 0}

DECL E6POS XP309={X 672,Y 199,Z 245,A 0,B 0,C 180,S 6,T 16,E1 0.0,E2 0.0,E3 0.0,E4 0.0,E5 0.0,E6 0.0}
DECL FDAT FP309={TOOL_NO 4,BASE_NO 0,IPO_FRAME #BASE,POINT2[] " "}
DECL LDAT LCPDAT309={VEL 1,ACC 50.000,APO_DIST 500.000,APO_FAC 50.0000,AXIS_VEL 50.000,AXIS_ACC 50.000,ORI_TYP #VAR,CIRC_TYP #BASE,JERK_FAC 50.0000,GEAR_JERK 100.000,EXAX_IGN 0}

DECL E6POS XP310={X 672,Y 249,Z 245,A 0,B 0,C 180,S 6,T 16,E1 0.0,E2 0.0,E3 0.0,E4 0.0,E5 0.0,E6 0.0}
DECL FDAT FP310={TOOL_NO 4,BASE_NO 0,IPO_FRAME #BASE,POINT2[] " "}
DECL LDAT LCPDAT310={VEL 1,ACC 50.000,APO_DIST 500.000,APO_FAC 50.0000,AXIS_VEL 50.000,AXIS_ACC 50.000,ORI_TYP #VAR,CIRC_TYP #BASE,JERK_FAC 50.0000,GEAR_JERK 100.000,EXAX_IGN 0}

DECL E6POS XP311={X 672,Y 299,Z 245,A 0,B 0,C 180,S 6,T 16,E1 0.0,E2 0.0,E3 0.0,E4 0.0,E5 0.0,E6 0.0}
DECL FDAT FP311={TOOL_NO 4,BASE_NO 0,IPO_FRAME #BASE,POINT2[] " "}
DECL LDAT LCPDAT311={VEL 1,ACC 50.000,APO_DIST 500.000,APO_FAC 50.0000,AXIS_VEL 50.000,AXIS_ACC 50.000,ORI_TYP #VAR,CIRC_TYP #BASE,JERK_FAC 50.0000,GEAR_JERK 100.000,EXAX_IGN 0}

DECL E6POS XP312={X 672,Y 349,Z 245,A 0,B 0,C 180,S 6,T 16,E1 0.0,E2 0.0,E3 0.0,E4 0.0,E5 0.0,E6 0.0}
DECL FDAT FP312={TOOL_NO 4,BASE_NO 0,IPO_FRAME #BASE,POINT2[] " "}
DECL LDAT LCPDAT312={VEL 1,ACC 50.000,APO_DIST 500.000,APO_FAC 50.0000,AXIS_VEL 50.000,AXIS_ACC 50.000,ORI_TYP #VAR,CIRC_TYP #BASE,JERK_FAC 50.0000,GEAR_JERK 100.000,EXAX_IGN 0}

DECL E6POS XP313={X 672,Y 399,Z 245,A 0,B 0,C 180,S 6,T 16,E1 0.0,E2 0.0,E3 0.0,E4 0.0,E5 0.0,E6 0.0}
DECL FDAT FP313={TOOL_NO 4,BASE_NO 0,IPO_FRAME #BASE,POINT2[] " "}
DECL LDAT LCPDAT313={VEL 1,ACC 50.000,APO_DIST 500.000,APO_FAC 50.0000,AXIS_VEL 50.000,AXIS_ACC 50.000,ORI_TYP #VAR,CIRC_TYP #BASE,JERK_FAC 50.0000,GEAR_JERK 100.000,EXAX_IGN 0}

DECL E6POS XP314={X 672,Y 449,Z 245,A 0,B 0,C 180,S 6,T 16,E1 0.0,E2 0.0,E3 0.0,E4 0.0,E5 0.0,E6 0.0}
DECL FDAT FP314={TOOL_NO 4,BASE_NO 0,IPO_FRAME #BASE,POINT2[] " "}
DECL LDAT LCPDAT314={VEL 1,ACC 50.000,APO_DIST 500.000,APO_FAC 50.0000,AXIS_VEL 50.000,AXIS_ACC 50.000,ORI_TYP #VAR,CIRC_TYP #BASE,JERK_FAC 50.0000,GEAR_JERK 100.000,EXAX_IGN 0}

DECL E6POS XP315={X 672,Y 499,Z 245,A 0,B 0,C 180,S 6,T 16,E1 0.0,E2 0.0,E3 0.0,E4 0.0,E5 0.0,E6 0.0}
DECL FDAT FP315={TOOL_NO 4,BASE_NO 0,IPO_FRAME #BASE,POINT2[] " "}
DECL LDAT LCPDAT315={VEL 1,ACC 50.000,APO_DIST 500.000,APO_FAC 50.0000,AXIS_VEL 50.000,AXIS_ACC 50.000,ORI_TYP #VAR,CIRC_TYP #BASE,JERK_FAC 50.0000,GEAR_JERK 100.000,EXAX_IGN 0}

DECL E6POS XP316={X 672,Y -51,Z 445,A 0,B 0,C 180,S 6,T 16,E1 0.0,E2 0.0,E3 0.0,E4 0.0,E5 0.0,E6 0.0}
DECL FDAT FP316={TOOL_NO 4,BASE_NO 0,IPO_FRAME #BASE,POINT2[] " "}
DECL LDAT LCPDAT316={VEL 0.25,ACC 12.000,APO_DIST 500.000,APO_FAC 50.0000,AXIS_VEL 12.000,AXIS_ACC 12.000,ORI_TYP #VAR,CIRC_TYP #BASE,JERK_FAC 50.0000,GEAR_JERK 100.000,EXAX_IGN 0}

DECL E6POS XP317={X 1272,Y -51,Z 445,A 0,B -90,C 180,S 6,T 50,E1 0.0,E2 0.0,E3 0.0,E4 0.0,E5 0.0,E6 0.0}
DECL FDAT FP317={TOOL_NO 4,BASE_NO 0,IPO_FRAME #BASE,POINT2[] " "}
DECL PDAT PPDAT317={VEL 20.000,ACC 20.000,APO_DIST 500.000,APO_MODE #CDIS,GEAR_JERK 100.000,EXAX_IGN 0}

DECL E6POS XP318={X 1272,Y -651,Z 445,A 0,B -90,C 180,S 6,T 16,E1 0.0,E2 0.0,E3 0.0,E4 0.0,E5 0.0,E6 0.0}
DECL FDAT FP318={TOOL_NO 4,BASE_NO 0,IPO_FRAME #BASE,POINT2[] " "}
DECL LDAT LCPDAT318={VEL 0.25,ACC 12.000,APO_DIST 500.000,APO_FAC 50.0000,AXIS_VEL 12.000,AXIS_ACC 12.000,ORI_TYP #VAR,CIRC_TYP #BASE,JERK_FAC 50.0000,GEAR_JERK 100.000,EXAX_IGN 0}

DECL E6POS XP319={X 1272,Y -651,Z -355,A 0,B -90,C 180,S 6,T 16,E1 0.0,E2 0.0,E3 0.0,E4 0.0,E5 0.0,E6 0.0}
DECL FDAT FP319={TOOL_NO 4,BASE_NO 0,IPO_FRAME #BASE,POINT2[] " "}
DECL LDAT LCPDAT319={VEL 1,ACC 50.000,APO_DIST 500.000,APO_FAC 50.0000,AXIS_VEL 50.000,AXIS_ACC 50.000,ORI_TYP #VAR,CIRC_TYP #BASE,JERK_FAC 50.0000,GEAR_JERK 100.000,EXAX_IGN 0}

DECL E6POS XP320={X 1222,Y -651,Z -355,A 0,B -90,C 180,S 6,T 16,E1 0.0,E2 0.0,E3 0.0,E4 0.0,E5 0.0,E6 0.0}
DECL FDAT FP320={TOOL_NO 4,BASE_NO 0,IPO_FRAME #BASE,POINT2[] " "}
DECL LDAT LCPDAT320={VEL 1,ACC 50.000,APO_DIST 500.000,APO_FAC 50.0000,AXIS_VEL 50.000,AXIS_ACC 50.000,ORI_TYP #VAR,CIRC_TYP #BASE,JERK_FAC 50.0000,GEAR_JERK 100.000,EXAX_IGN 0}

DECL E6POS XP321={X 1172,Y -651,Z -355,A 0,B -90,C 180,S 6,T 16,E1 0.0,E2 0.0,E3 0.0,E4 0.0,E5 0.0,E6 0.0}
DECL FDAT FP321={TOOL_NO 4,BASE_NO 0,IPO_FRAME #BASE,POINT2[] " "}
DECL LDAT LCPDAT321={VEL 1,ACC 50.000,APO_DIST 500.000,APO_FAC 50.0000,AXIS_VEL 50.000,AXIS_ACC 50.000,ORI_TYP #VAR,CIRC_TYP #BASE,JERK_FAC 50.0000,GEAR_JERK 100.000,EXAX_IGN 0}

DECL E6POS XP322={X 1122,Y -651,Z -355,A 0,B -90,C 180,S 6,T 16,E1 0.0,E2 0.0,E3 0.0,E4 0.0,E5 0.0,E6 0.0}
DECL FDAT FP322={TOOL_NO 4,BASE_NO 0,IPO_FRAME #BASE,POINT2[] " "}
DECL LDAT LCPDAT322={VEL 1,ACC 50.000,APO_DIST 500.000,APO_FAC 50.0000,AXIS_VEL 50.000,AXIS_ACC 50.000,ORI_TYP #VAR,CIRC_TYP #BASE,JERK_FAC 50.0000,GEAR_JERK 100.000,EXAX_IGN 0}

DECL E6POS XP323={X 1072,Y -651,Z -355,A 0,B -90,C 180,S 6,T 16,E1 0.0,E2 0.0,E3 0.0,E4 0.0,E5 0.0,E6 0.0}
DECL FDAT FP323={TOOL_NO 4,BASE_NO 0,IPO_FRAME #BASE,POINT2[] " "}
DECL LDAT LCPDAT323={VEL 1,ACC 50.000,APO_DIST 500.000,APO_FAC 50.0000,AXIS_VEL 50.000,AXIS_ACC 50.000,ORI_TYP #VAR,CIRC_TYP #BASE,JERK_FAC 50.0000,GEAR_JERK 100.000,EXAX_IGN 0}

DECL E6POS XP324={X 1022,Y -651,Z -355,A 0,B -90,C 180,S 6,T 16,E1 0.0,E2 0.0,E3 0.0,E4 0.0,E5 0.0,E6 0.0}
DECL FDAT FP324={TOOL_NO 4,BASE_NO 0,IPO_FRAME #BASE,POINT2[] " "}
DECL LDAT LCPDAT324={VEL 1,ACC 50.000,APO_DIST 500.000,APO_FAC 50.0000,AXIS_VEL 50.000,AXIS_ACC 50.000,ORI_TYP #VAR,CIRC_TYP #BASE,JERK_FAC 50.0000,GEAR_JERK 100.000,EXAX_IGN 0}

DECL E6POS XP325={X 972,Y -651,Z -355,A 0,B -90,C 180,S 6,T 16,E1 0.0,E2 0.0,E3 0.0,E4 0.0,E5 0.0,E6 0.0}
DECL FDAT FP325={TOOL_NO 4,BASE_NO 0,IPO_FRAME #BASE,POINT2[] " "}
DECL LDAT LCPDAT325={VEL 1,ACC 50.000,APO_DIST 500.000,APO_FAC 50.0000,AXIS_VEL 50.000,AXIS_ACC 50.000,ORI_TYP #VAR,CIRC_TYP #BASE,JERK_FAC 50.0000,GEAR_JERK 100.000,EXAX_IGN 0}

DECL E6POS XP326={X 922,Y -651,Z -355,A 0,B -90,C 180,S 6,T 16,E1 0.0,E2 0.0,E3 0.0,E4 0.0,E5 0.0,E6 0.0}
DECL FDAT FP326={TOOL_NO 4,BASE_NO 0,IPO_FRAME #BASE,POINT2[] " "}
DECL LDAT LCPDAT326={VEL 1,ACC 50.000,APO_DIST 500.000,APO_FAC 50.0000,AXIS_VEL 50.000,AXIS_ACC 50.000,ORI_TYP #VAR,CIRC_TYP #BASE,JERK_FAC 50.0000,GEAR_JERK 100.000,EXAX_IGN 0}

DECL E6POS XP327={X 872,Y -651,Z -355,A 0,B -90,C 180,S 6,T 16,E1 0.0,E2 0.0,E3 0.0,E4 0.0,E5 0.0,E6 0.0}
DECL FDAT FP327={TOOL_NO 4,BASE_NO 0,IPO_FRAME #BASE,POINT2[] " "}
DECL LDAT LCPDAT327={VEL 1,ACC 50.000,APO_DIST 500.000,APO_FAC 50.0000,AXIS_VEL 50.000,AXIS_ACC 50.000,ORI_TYP #VAR,CIRC_TYP #BASE,JERK_FAC 50.0000,GEAR_JERK 100.000,EXAX_IGN 0}

DECL E6POS XP328={X 822,Y -651,Z -355,A 0,B -90,C 180,S 6,T 16,E1 0.0,E2 0.0,E3 0.0,E4 0.0,E5 0.0,E6 0.0}
DECL FDAT FP328={TOOL_NO 4,BASE_NO 0,IPO_FRAME #BASE,POINT2[] " "}
DECL LDAT LCPDAT328={VEL 1,ACC 50.000,APO_DIST 500.000,APO_FAC 50.0000,AXIS_VEL 50.000,AXIS_ACC 50.000,ORI_TYP #VAR,CIRC_TYP #BASE,JERK_FAC 50.0000,GEAR_JERK 100.000,EXAX_IGN 0}

DECL E6POS XP329={X 772,Y -651,Z -355,A 0,B -90,C 180,S 6,T 16,E1 0.0,E2 0.0,E3 0.0,E4 0.0,E5 0.0,E6 0.0}
DECL FDAT FP329={TOOL_NO 4,BASE_NO 0,IPO_FRAME #BASE,POINT2[] " "}
DECL LDAT LCPDAT329={VEL 1,ACC 50.000,APO_DIST 500.000,APO_FAC 50.0000,AXIS_VEL 50.000,AXIS_ACC 50.000,ORI_TYP #VAR,CIRC_TYP #BASE,JERK_FAC 50.0000,GEAR_JERK 100.000,EXAX_IGN 0}

DECL E6POS XP330={X 722,Y -651,Z -355,A 0,B -90,C 180,S 6,T 16,E1 0.0,E2 0.0,E3 0.0,E4 0.0,E5 0.0,E6 0.0}
DECL FDAT FP330={TOOL_NO 4,BASE_NO 0,IPO_FRAME #BASE,POINT2[] " "}
DECL LDAT LCPDAT330={VEL 1,ACC 50.000,APO_DIST 500.000,APO_FAC 50.0000,AXIS_VEL 50.000,AXIS_ACC 50.000,ORI_TYP #VAR,CIRC_TYP #BASE,JERK_FAC 50.0000,GEAR_JERK 100.000,EXAX_IGN 0}

DECL E6POS XP331={X 672,Y -651,Z -355,A 0,B -90,C 180,S 6,T 16,E1 0.0,E2 0.0,E3 0.0,E4 0.0,E5 0.0,E6 0.0}
DECL FDAT FP331={TOOL_NO 4,BASE_NO 0,IPO_FRAME #BASE,POINT2[] " "}
DECL LDAT LCPDAT331={VEL 1,ACC 50.000,APO_DIST 500.000,APO_FAC 50.0000,AXIS_VEL 50.000,AXIS_ACC 50.000,ORI_TYP #VAR,CIRC_TYP #BASE,JERK_FAC 50.0000,GEAR_JERK 100.000,EXAX_IGN 0}

DECL E6POS XP332={X 672,Y -651,Z -305,A 0,B -90,C 180,S 6,T 16,E1 0.0,E2 0.0,E3 0.0,E4 0.0,E5 0.0,E6 0.0}
DECL FDAT FP332={TOOL_NO 4,BASE_NO 0,IPO_FRAME #BASE,POINT2[] " "}
DECL LDAT LCPDAT332={VEL 1,ACC 50.000,APO_DIST 500.000,APO_FAC 50.0000,AXIS_VEL 50.000,AXIS_ACC 50.000,ORI_TYP #VAR,CIRC_TYP #BASE,JERK_FAC 50.0000,GEAR_JERK 100.000,EXAX_IGN 0}

DECL E6POS XP333={X 722,Y -651,Z -305,A 0,B -90,C 180,S 6,T 16,E1 0.0,E2 0.0,E3 0.0,E4 0.0,E5 0.0,E6 0.0}
DECL FDAT FP333={TOOL_NO 4,BASE_NO 0,IPO_FRAME #BASE,POINT2[] " "}
DECL LDAT LCPDAT333={VEL 1,ACC 50.000,APO_DIST 500.000,APO_FAC 50.0000,AXIS_VEL 50.000,AXIS_ACC 50.000,ORI_TYP #VAR,CIRC_TYP #BASE,JERK_FAC 50.0000,GEAR_JERK 100.000,EXAX_IGN 0}

DECL E6POS XP334={X 772,Y -651,Z -305,A 0,B -90,C 180,S 6,T 16,E1 0.0,E2 0.0,E3 0.0,E4 0.0,E5 0.0,E6 0.0}
DECL FDAT FP334={TOOL_NO 4,BASE_NO 0,IPO_FRAME #BASE,POINT2[] " "}
DECL LDAT LCPDAT334={VEL 1,ACC 50.000,APO_DIST 500.000,APO_FAC 50.0000,AXIS_VEL 50.000,AXIS_ACC 50.000,ORI_TYP #VAR,CIRC_TYP #BASE,JERK_FAC 50.0000,GEAR_JERK 100.000,EXAX_IGN 0}

DECL E6POS XP335={X 822,Y -651,Z -305,A 0,B -90,C 180,S 6,T 16,E1 0.0,E2 0.0,E3 0.0,E4 0.0,E5 0.0,E6 0.0}
DECL FDAT FP335={TOOL_NO 4,BASE_NO 0,IPO_FRAME #BASE,POINT2[] " "}
DECL LDAT LCPDAT335={VEL 1,ACC 50.000,APO_DIST 500.000,APO_FAC 50.0000,AXIS_VEL 50.000,AXIS_ACC 50.000,ORI_TYP #VAR,CIRC_TYP #BASE,JERK_FAC 50.0000,GEAR_JERK 100.000,EXAX_IGN 0}

DECL E6POS XP336={X 872,Y -651,Z -305,A 0,B -90,C 180,S 6,T 16,E1 0.0,E2 0.0,E3 0.0,E4 0.0,E5 0.0,E6 0.0}
DECL FDAT FP336={TOOL_NO 4,BASE_NO 0,IPO_FRAME #BASE,POINT2[] " "}
DECL LDAT LCPDAT336={VEL 1,ACC 50.000,APO_DIST 500.000,APO_FAC 50.0000,AXIS_VEL 50.000,AXIS_ACC 50.000,ORI_TYP #VAR,CIRC_TYP #BASE,JERK_FAC 50.0000,GEAR_JERK 100.000,EXAX_IGN 0}

DECL E6POS XP337={X 922,Y -651,Z -305,A 0,B -90,C 180,S 6,T 16,E1 0.0,E2 0.0,E3 0.0,E4 0.0,E5 0.0,E6 0.0}
DECL FDAT FP337={TOOL_NO 4,BASE_NO 0,IPO_FRAME #BASE,POINT2[] " "}
DECL LDAT LCPDAT337={VEL 1,ACC 50.000,APO_DIST 500.000,APO_FAC 50.0000,AXIS_VEL 50.000,AXIS_ACC 50.000,ORI_TYP #VAR,CIRC_TYP #BASE,JERK_FAC 50.0000,GEAR_JERK 100.000,EXAX_IGN 0}

DECL E6POS XP338={X 972,Y -651,Z -305,A 0,B -90,C 180,S 6,T 16,E1 0.0,E2 0.0,E3 0.0,E4 0.0,E5 0.0,E6 0.0}
DECL FDAT FP338={TOOL_NO 4,BASE_NO 0,IPO_FRAME #BASE,POINT2[] " "}
DECL LDAT LCPDAT338={VEL 1,ACC 50.000,APO_DIST 500.000,APO_FAC 50.0000,AXIS_VEL 50.000,AXIS_ACC 50.000,ORI_TYP #VAR,CIRC_TYP #BASE,JERK_FAC 50.0000,GEAR_JERK 100.000,EXAX_IGN 0}

DECL E6POS XP339={X 1022,Y -651,Z -305,A 0,B -90,C 180,S 6,T 16,E1 0.0,E2 0.0,E3 0.0,E4 0.0,E5 0.0,E6 0.0}
DECL FDAT FP339={TOOL_NO 4,BASE_NO 0,IPO_FRAME #BASE,POINT2[] " "}
DECL LDAT LCPDAT339={VEL 1,ACC 50.000,APO_DIST 500.000,APO_FAC 50.0000,AXIS_VEL 50.000,AXIS_ACC 50.000,ORI_TYP #VAR,CIRC_TYP #BASE,JERK_FAC 50.0000,GEAR_JERK 100.000,EXAX_IGN 0}

DECL E6POS XP340={X 1072,Y -651,Z -305,A 0,B -90,C 180,S 6,T 16,E1 0.0,E2 0.0,E3 0.0,E4 0.0,E5 0.0,E6 0.0}
DECL FDAT FP340={TOOL_NO 4,BASE_NO 0,IPO_FRAME #BASE,POINT2[] " "}
DECL LDAT LCPDAT340={VEL 1,ACC 50.000,APO_DIST 500.000,APO_FAC 50.0000,AXIS_VEL 50.000,AXIS_ACC 50.000,ORI_TYP #VAR,CIRC_TYP #BASE,JERK_FAC 50.0000,GEAR_JERK 100.000,EXAX_IGN 0}

DECL E6POS XP341={X 1122,Y -651,Z -305,A 0,B -90,C 180,S 6,T 16,E1 0.0,E2 0.0,E3 0.0,E4 0.0,E5 0.0,E6 0.0}
DECL FDAT FP341={TOOL_NO 4,BASE_NO 0,IPO_FRAME #BASE,POINT2[] " "}
DECL LDAT LCPDAT341={VEL 1,ACC 50.000,APO_DIST 500.000,APO_FAC 50.0000,AXIS_VEL 50.000,AXIS_ACC 50.000,ORI_TYP #VAR,CIRC_TYP #BASE,JERK_FAC 50.0000,GEAR_JERK 100.000,EXAX_IGN 0}

DECL E6POS XP342={X 1172,Y -651,Z -305,A 0,B -90,C 180,S 6,T 16,E1 0.0,E2 0.0,E3 0.0,E4 0.0,E5 0.0,E6 0.0}
DECL FDAT FP342={TOOL_NO 4,BASE_NO 0,IPO_FRAME #BASE,POINT2[] " "}
DECL LDAT LCPDAT342={VEL 1,ACC 50.000,APO_DIST 500.000,APO_FAC 50.0000,AXIS_VEL 50.000,AXIS_ACC 50.000,ORI_TYP #VAR,CIRC_TYP #BASE,JERK_FAC 50.0000,GEAR_JERK 100.000,EXAX_IGN 0}

DECL E6POS XP343={X 1222,Y -651,Z -305,A 0,B -90,C 180,S 6,T 16,E1 0.0,E2 0.0,E3 0.0,E4 0.0,E5 0.0,E6 0.0}
DECL FDAT FP343={TOOL_NO 4,BASE_NO 0,IPO_FRAME #BASE,POINT2[] " "}
DECL LDAT LCPDAT343={VEL 1,ACC 50.000,APO_DIST 500.000,APO_FAC 50.0000,AXIS_VEL 50.000,AXIS_ACC 50.000,ORI_TYP #VAR,CIRC_TYP #BASE,JERK_FAC 50.0000,GEAR_JERK 100.000,EXAX_IGN 0}

DECL E6POS XP344={X 1272,Y -651,Z -305,A 0,B -90,C 180,S 6,T 16,E1 0.0,E2 0.0,E3 0.0,E4 0.0,E5 0.0,E6 0.0}
DECL FDAT FP344={TOOL_NO 4,BASE_NO 0,IPO_FRAME #BASE,POINT2[] " "}
DECL LDAT LCPDAT344={VEL 1,ACC 50.000,APO_DIST 500.000,APO_FAC 50.0000,AXIS_VEL 50.000,AXIS_ACC 50.000,ORI_TYP #VAR,CIRC_TYP #BASE,JERK_FAC 50.0000,GEAR_JERK 100.000,EXAX_IGN 0}

DECL E6POS XP345={X 1272,Y -651,Z -255,A 0,B -90,C 180,S 6,T 16,E1 0.0,E2 0.0,E3 0.0,E4 0.0,E5 0.0,E6 0.0}
DECL FDAT FP345={TOOL_NO 4,BASE_NO 0,IPO_FRAME #BASE,POINT2[] " "}
DECL LDAT LCPDAT345={VEL 1,ACC 50.000,APO_DIST 500.000,APO_FAC 50.0000,AXIS_VEL 50.000,AXIS_ACC 50.000,ORI_TYP #VAR,CIRC_TYP #BASE,JERK_FAC 50.0000,GEAR_JERK 100.000,EXAX_IGN 0}

DECL E6POS XP346={X 1222,Y -651,Z -255,A 0,B -90,C 180,S 6,T 16,E1 0.0,E2 0.0,E3 0.0,E4 0.0,E5 0.0,E6 0.0}
DECL FDAT FP346={TOOL_NO 4,BASE_NO 0,IPO_FRAME #BASE,POINT2[] " "}
DECL LDAT LCPDAT346={VEL 1,ACC 50.000,APO_DIST 500.000,APO_FAC 50.0000,AXIS_VEL 50.000,AXIS_ACC 50.000,ORI_TYP #VAR,CIRC_TYP #BASE,JERK_FAC 50.0000,GEAR_JERK 100.000,EXAX_IGN 0}

DECL E6POS XP347={X 1172,Y -651,Z -255,A 0,B -90,C 180,S 6,T 16,E1 0.0,E2 0.0,E3 0.0,E4 0.0,E5 0.0,E6 0.0}
DECL FDAT FP347={TOOL_NO 4,BASE_NO 0,IPO_FRAME #BASE,POINT2[] " "}
DECL LDAT LCPDAT347={VEL 1,ACC 50.000,APO_DIST 500.000,APO_FAC 50.0000,AXIS_VEL 50.000,AXIS_ACC 50.000,ORI_TYP #VAR,CIRC_TYP #BASE,JERK_FAC 50.0000,GEAR_JERK 100.000,EXAX_IGN 0}

DECL E6POS XP348={X 1122,Y -651,Z -255,A 0,B -90,C 180,S 6,T 16,E1 0.0,E2 0.0,E3 0.0,E4 0.0,E5 0.0,E6 0.0}
DECL FDAT FP348={TOOL_NO 4,BASE_NO 0,IPO_FRAME #BASE,POINT2[] " "}
DECL LDAT LCPDAT348={VEL 1,ACC 50.000,APO_DIST 500.000,APO_FAC 50.0000,AXIS_VEL 50.000,AXIS_ACC 50.000,ORI_TYP #VAR,CIRC_TYP #BASE,JERK_FAC 50.0000,GEAR_JERK 100.000,EXAX_IGN 0}

DECL E6POS XP349={X 1072,Y -651,Z -255,A 0,B -90,C 180,S 6,T 16,E1 0.0,E2 0.0,E3 0.0,E4 0.0,E5 0.0,E6 0.0}
DECL FDAT FP349={TOOL_NO 4,BASE_NO 0,IPO_FRAME #BASE,POINT2[] " "}
DECL LDAT LCPDAT349={VEL 1,ACC 50.000,APO_DIST 500.000,APO_FAC 50.0000,AXIS_VEL 50.000,AXIS_ACC 50.000,ORI_TYP #VAR,CIRC_TYP #BASE,JERK_FAC 50.0000,GEAR_JERK 100.000,EXAX_IGN 0}

DECL E6POS XP350={X 1022,Y -651,Z -255,A 0,B -90,C 180,S 6,T 16,E1 0.0,E2 0.0,E3 0.0,E4 0.0,E5 0.0,E6 0.0}
DECL FDAT FP350={TOOL_NO 4,BASE_NO 0,IPO_FRAME #BASE,POINT2[] " "}
DECL LDAT LCPDAT350={VEL 1,ACC 50.000,APO_DIST 500.000,APO_FAC 50.0000,AXIS_VEL 50.000,AXIS_ACC 50.000,ORI_TYP #VAR,CIRC_TYP #BASE,JERK_FAC 50.0000,GEAR_JERK 100.000,EXAX_IGN 0}

DECL E6POS XP351={X 972,Y -651,Z -255,A 0,B -90,C 180,S 6,T 16,E1 0.0,E2 0.0,E3 0.0,E4 0.0,E5 0.0,E6 0.0}
DECL FDAT FP351={TOOL_NO 4,BASE_NO 0,IPO_FRAME #BASE,POINT2[] " "}
DECL LDAT LCPDAT351={VEL 1,ACC 50.000,APO_DIST 500.000,APO_FAC 50.0000,AXIS_VEL 50.000,AXIS_ACC 50.000,ORI_TYP #VAR,CIRC_TYP #BASE,JERK_FAC 50.0000,GEAR_JERK 100.000,EXAX_IGN 0}

DECL E6POS XP352={X 922,Y -651,Z -255,A 0,B -90,C 180,S 6,T 16,E1 0.0,E2 0.0,E3 0.0,E4 0.0,E5 0.0,E6 0.0}
DECL FDAT FP352={TOOL_NO 4,BASE_NO 0,IPO_FRAME #BASE,POINT2[] " "}
DECL LDAT LCPDAT352={VEL 1,ACC 50.000,APO_DIST 500.000,APO_FAC 50.0000,AXIS_VEL 50.000,AXIS_ACC 50.000,ORI_TYP #VAR,CIRC_TYP #BASE,JERK_FAC 50.0000,GEAR_JERK 100.000,EXAX_IGN 0}

DECL E6POS XP353={X 872,Y -651,Z -255,A 0,B -90,C 180,S 6,T 16,E1 0.0,E2 0.0,E3 0.0,E4 0.0,E5 0.0,E6 0.0}
DECL FDAT FP353={TOOL_NO 4,BASE_NO 0,IPO_FRAME #BASE,POINT2[] " "}
DECL LDAT LCPDAT353={VEL 1,ACC 50.000,APO_DIST 500.000,APO_FAC 50.0000,AXIS_VEL 50.000,AXIS_ACC 50.000,ORI_TYP #VAR,CIRC_TYP #BASE,JERK_FAC 50.0000,GEAR_JERK 100.000,EXAX_IGN 0}

DECL E6POS XP354={X 822,Y -651,Z -255,A 0,B -90,C 180,S 6,T 16,E1 0.0,E2 0.0,E3 0.0,E4 0.0,E5 0.0,E6 0.0}
DECL FDAT FP354={TOOL_NO 4,BASE_NO 0,IPO_FRAME #BASE,POINT2[] " "}
DECL LDAT LCPDAT354={VEL 1,ACC 50.000,APO_DIST 500.000,APO_FAC 50.0000,AXIS_VEL 50.000,AXIS_ACC 50.000,ORI_TYP #VAR,CIRC_TYP #BASE,JERK_FAC 50.0000,GEAR_JERK 100.000,EXAX_IGN 0}

DECL E6POS XP355={X 772,Y -651,Z -255,A 0,B -90,C 180,S 6,T 16,E1 0.0,E2 0.0,E3 0.0,E4 0.0,E5 0.0,E6 0.0}
DECL FDAT FP355={TOOL_NO 4,BASE_NO 0,IPO_FRAME #BASE,POINT2[] " "}
DECL LDAT LCPDAT355={VEL 1,ACC 50.000,APO_DIST 500.000,APO_FAC 50.0000,AXIS_VEL 50.000,AXIS_ACC 50.000,ORI_TYP #VAR,CIRC_TYP #BASE,JERK_FAC 50.0000,GEAR_JERK 100.000,EXAX_IGN 0}

DECL E6POS XP356={X 722,Y -651,Z -255,A 0,B -90,C 180,S 6,T 16,E1 0.0,E2 0.0,E3 0.0,E4 0.0,E5 0.0,E6 0.0}
DECL FDAT FP356={TOOL_NO 4,BASE_NO 0,IPO_FRAME #BASE,POINT2[] " "}
DECL LDAT LCPDAT356={VEL 1,ACC 50.000,APO_DIST 500.000,APO_FAC 50.0000,AXIS_VEL 50.000,AXIS_ACC 50.000,ORI_TYP #VAR,CIRC_TYP #BASE,JERK_FAC 50.0000,GEAR_JERK 100.000,EXAX_IGN 0}

DECL E6POS XP357={X 672,Y -651,Z -255,A 0,B -90,C 180,S 6,T 16,E1 0.0,E2 0.0,E3 0.0,E4 0.0,E5 0.0,E6 0.0}
DECL FDAT FP357={TOOL_NO 4,BASE_NO 0,IPO_FRAME #BASE,POINT2[] " "}
DECL LDAT LCPDAT357={VEL 1,ACC 50.000,APO_DIST 500.000,APO_FAC 50.0000,AXIS_VEL 50.000,AXIS_ACC 50.000,ORI_TYP #VAR,CIRC_TYP #BASE,JERK_FAC 50.0000,GEAR_JERK 100.000,EXAX_IGN 0}

DECL E6POS XP358={X 672,Y -651,Z -205,A 0,B -90,C 180,S 6,T 16,E1 0.0,E2 0.0,E3 0.0,E4 0.0,E5 0.0,E6 0.0}
DECL FDAT FP358={TOOL_NO 4,BASE_NO 0,IPO_FRAME #BASE,POINT2[] " "}
DECL LDAT LCPDAT358={VEL 1,ACC 50.000,APO_DIST 500.000,APO_FAC 50.0000,AXIS_VEL 50.000,AXIS_ACC 50.000,ORI_TYP #VAR,CIRC_TYP #BASE,JERK_FAC 50.0000,GEAR_JERK 100.000,EXAX_IGN 0}

DECL E6POS XP359={X 722,Y -651,Z -205,A 0,B -90,C 180,S 6,T 16,E1 0.0,E2 0.0,E3 0.0,E4 0.0,E5 0.0,E6 0.0}
DECL FDAT FP359={TOOL_NO 4,BASE_NO 0,IPO_FRAME #BASE,POINT2[] " "}
DECL LDAT LCPDAT359={VEL 1,ACC 50.000,APO_DIST 500.000,APO_FAC 50.0000,AXIS_VEL 50.000,AXIS_ACC 50.000,ORI_TYP #VAR,CIRC_TYP #BASE,JERK_FAC 50.0000,GEAR_JERK 100.000,EXAX_IGN 0}

DECL E6POS XP360={X 772,Y -651,Z -205,A 0,B -90,C 180,S 6,T 16,E1 0.0,E2 0.0,E3 0.0,E4 0.0,E5 0.0,E6 0.0}
DECL FDAT FP360={TOOL_NO 4,BASE_NO 0,IPO_FRAME #BASE,POINT2[] " "}
DECL LDAT LCPDAT360={VEL 1,ACC 50.000,APO_DIST 500.000,APO_FAC 50.0000,AXIS_VEL 50.000,AXIS_ACC 50.000,ORI_TYP #VAR,CIRC_TYP #BASE,JERK_FAC 50.0000,GEAR_JERK 100.000,EXAX_IGN 0}

DECL E6POS XP361={X 822,Y -651,Z -205,A 0,B -90,C 180,S 6,T 16,E1 0.0,E2 0.0,E3 0.0,E4 0.0,E5 0.0,E6 0.0}
DECL FDAT FP361={TOOL_NO 4,BASE_NO 0,IPO_FRAME #BASE,POINT2[] " "}
DECL LDAT LCPDAT361={VEL 1,ACC 50.000,APO_DIST 500.000,APO_FAC 50.0000,AXIS_VEL 50.000,AXIS_ACC 50.000,ORI_TYP #VAR,CIRC_TYP #BASE,JERK_FAC 50.0000,GEAR_JERK 100.000,EXAX_IGN 0}

DECL E6POS XP362={X 872,Y -651,Z -205,A 0,B -90,C 180,S 6,T 16,E1 0.0,E2 0.0,E3 0.0,E4 0.0,E5 0.0,E6 0.0}
DECL FDAT FP362={TOOL_NO 4,BASE_NO 0,IPO_FRAME #BASE,POINT2[] " "}
DECL LDAT LCPDAT362={VEL 1,ACC 50.000,APO_DIST 500.000,APO_FAC 50.0000,AXIS_VEL 50.000,AXIS_ACC 50.000,ORI_TYP #VAR,CIRC_TYP #BASE,JERK_FAC 50.0000,GEAR_JERK 100.000,EXAX_IGN 0}

DECL E6POS XP363={X 922,Y -651,Z -205,A 0,B -90,C 180,S 6,T 16,E1 0.0,E2 0.0,E3 0.0,E4 0.0,E5 0.0,E6 0.0}
DECL FDAT FP363={TOOL_NO 4,BASE_NO 0,IPO_FRAME #BASE,POINT2[] " "}
DECL LDAT LCPDAT363={VEL 1,ACC 50.000,APO_DIST 500.000,APO_FAC 50.0000,AXIS_VEL 50.000,AXIS_ACC 50.000,ORI_TYP #VAR,CIRC_TYP #BASE,JERK_FAC 50.0000,GEAR_JERK 100.000,EXAX_IGN 0}

DECL E6POS XP364={X 972,Y -651,Z -205,A 0,B -90,C 180,S 6,T 16,E1 0.0,E2 0.0,E3 0.0,E4 0.0,E5 0.0,E6 0.0}
DECL FDAT FP364={TOOL_NO 4,BASE_NO 0,IPO_FRAME #BASE,POINT2[] " "}
DECL LDAT LCPDAT364={VEL 1,ACC 50.000,APO_DIST 500.000,APO_FAC 50.0000,AXIS_VEL 50.000,AXIS_ACC 50.000,ORI_TYP #VAR,CIRC_TYP #BASE,JERK_FAC 50.0000,GEAR_JERK 100.000,EXAX_IGN 0}

DECL E6POS XP365={X 1022,Y -651,Z -205,A 0,B -90,C 180,S 6,T 16,E1 0.0,E2 0.0,E3 0.0,E4 0.0,E5 0.0,E6 0.0}
DECL FDAT FP365={TOOL_NO 4,BASE_NO 0,IPO_FRAME #BASE,POINT2[] " "}
DECL LDAT LCPDAT365={VEL 1,ACC 50.000,APO_DIST 500.000,APO_FAC 50.0000,AXIS_VEL 50.000,AXIS_ACC 50.000,ORI_TYP #VAR,CIRC_TYP #BASE,JERK_FAC 50.0000,GEAR_JERK 100.000,EXAX_IGN 0}

DECL E6POS XP366={X 1072,Y -651,Z -205,A 0,B -90,C 180,S 6,T 16,E1 0.0,E2 0.0,E3 0.0,E4 0.0,E5 0.0,E6 0.0}
DECL FDAT FP366={TOOL_NO 4,BASE_NO 0,IPO_FRAME #BASE,POINT2[] " "}
DECL LDAT LCPDAT366={VEL 1,ACC 50.000,APO_DIST 500.000,APO_FAC 50.0000,AXIS_VEL 50.000,AXIS_ACC 50.000,ORI_TYP #VAR,CIRC_TYP #BASE,JERK_FAC 50.0000,GEAR_JERK 100.000,EXAX_IGN 0}

DECL E6POS XP367={X 1122,Y -651,Z -205,A 0,B -90,C 180,S 6,T 16,E1 0.0,E2 0.0,E3 0.0,E4 0.0,E5 0.0,E6 0.0}
DECL FDAT FP367={TOOL_NO 4,BASE_NO 0,IPO_FRAME #BASE,POINT2[] " "}
DECL LDAT LCPDAT367={VEL 1,ACC 50.000,APO_DIST 500.000,APO_FAC 50.0000,AXIS_VEL 50.000,AXIS_ACC 50.000,ORI_TYP #VAR,CIRC_TYP #BASE,JERK_FAC 50.0000,GEAR_JERK 100.000,EXAX_IGN 0}

DECL E6POS XP368={X 1172,Y -651,Z -205,A 0,B -90,C 180,S 6,T 16,E1 0.0,E2 0.0,E3 0.0,E4 0.0,E5 0.0,E6 0.0}
DECL FDAT FP368={TOOL_NO 4,BASE_NO 0,IPO_FRAME #BASE,POINT2[] " "}
DECL LDAT LCPDAT368={VEL 1,ACC 50.000,APO_DIST 500.000,APO_FAC 50.0000,AXIS_VEL 50.000,AXIS_ACC 50.000,ORI_TYP #VAR,CIRC_TYP #BASE,JERK_FAC 50.0000,GEAR_JERK 100.000,EXAX_IGN 0}

DECL E6POS XP369={X 1222,Y -651,Z -205,A 0,B -90,C 180,S 6,T 16,E1 0.0,E2 0.0,E3 0.0,E4 0.0,E5 0.0,E6 0.0}
DECL FDAT FP369={TOOL_NO 4,BASE_NO 0,IPO_FRAME #BASE,POINT2[] " "}
DECL LDAT LCPDAT369={VEL 1,ACC 50.000,APO_DIST 500.000,APO_FAC 50.0000,AXIS_VEL 50.000,AXIS_ACC 50.000,ORI_TYP #VAR,CIRC_TYP #BASE,JERK_FAC 50.0000,GEAR_JERK 100.000,EXAX_IGN 0}

DECL E6POS XP370={X 1272,Y -651,Z -205,A 0,B -90,C 180,S 6,T 16,E1 0.0,E2 0.0,E3 0.0,E4 0.0,E5 0.0,E6 0.0}
DECL FDAT FP370={TOOL_NO 4,BASE_NO 0,IPO_FRAME #BASE,POINT2[] " "}
DECL LDAT LCPDAT370={VEL 1,ACC 50.000,APO_DIST 500.000,APO_FAC 50.0000,AXIS_VEL 50.000,AXIS_ACC 50.000,ORI_TYP #VAR,CIRC_TYP #BASE,JERK_FAC 50.0000,GEAR_JERK 100.000,EXAX_IGN 0}

DECL E6POS XP371={X 1272,Y -651,Z -155,A 0,B -90,C 180,S 6,T 16,E1 0.0,E2 0.0,E3 0.0,E4 0.0,E5 0.0,E6 0.0}
DECL FDAT FP371={TOOL_NO 4,BASE_NO 0,IPO_FRAME #BASE,POINT2[] " "}
DECL LDAT LCPDAT371={VEL 1,ACC 50.000,APO_DIST 500.000,APO_FAC 50.0000,AXIS_VEL 50.000,AXIS_ACC 50.000,ORI_TYP #VAR,CIRC_TYP #BASE,JERK_FAC 50.0000,GEAR_JERK 100.000,EXAX_IGN 0}

DECL E6POS XP372={X 1222,Y -651,Z -155,A 0,B -90,C 180,S 6,T 16,E1 0.0,E2 0.0,E3 0.0,E4 0.0,E5 0.0,E6 0.0}
DECL FDAT FP372={TOOL_NO 4,BASE_NO 0,IPO_FRAME #BASE,POINT2[] " "}
DECL LDAT LCPDAT372={VEL 1,ACC 50.000,APO_DIST 500.000,APO_FAC 50.0000,AXIS_VEL 50.000,AXIS_ACC 50.000,ORI_TYP #VAR,CIRC_TYP #BASE,JERK_FAC 50.0000,GEAR_JERK 100.000,EXAX_IGN 0}

DECL E6POS XP373={X 1172,Y -651,Z -155,A 0,B -90,C 180,S 6,T 16,E1 0.0,E2 0.0,E3 0.0,E4 0.0,E5 0.0,E6 0.0}
DECL FDAT FP373={TOOL_NO 4,BASE_NO 0,IPO_FRAME #BASE,POINT2[] " "}
DECL LDAT LCPDAT373={VEL 1,ACC 50.000,APO_DIST 500.000,APO_FAC 50.0000,AXIS_VEL 50.000,AXIS_ACC 50.000,ORI_TYP #VAR,CIRC_TYP #BASE,JERK_FAC 50.0000,GEAR_JERK 100.000,EXAX_IGN 0}

DECL E6POS XP374={X 1122,Y -651,Z -155,A 0,B -90,C 180,S 6,T 16,E1 0.0,E2 0.0,E3 0.0,E4 0.0,E5 0.0,E6 0.0}
DECL FDAT FP374={TOOL_NO 4,BASE_NO 0,IPO_FRAME #BASE,POINT2[] " "}
DECL LDAT LCPDAT374={VEL 1,ACC 50.000,APO_DIST 500.000,APO_FAC 50.0000,AXIS_VEL 50.000,AXIS_ACC 50.000,ORI_TYP #VAR,CIRC_TYP #BASE,JERK_FAC 50.0000,GEAR_JERK 100.000,EXAX_IGN 0}

DECL E6POS XP375={X 1072,Y -651,Z -155,A 0,B -90,C 180,S 6,T 16,E1 0.0,E2 0.0,E3 0.0,E4 0.0,E5 0.0,E6 0.0}
DECL FDAT FP375={TOOL_NO 4,BASE_NO 0,IPO_FRAME #BASE,POINT2[] " "}
DECL LDAT LCPDAT375={VEL 1,ACC 50.000,APO_DIST 500.000,APO_FAC 50.0000,AXIS_VEL 50.000,AXIS_ACC 50.000,ORI_TYP #VAR,CIRC_TYP #BASE,JERK_FAC 50.0000,GEAR_JERK 100.000,EXAX_IGN 0}

DECL E6POS XP376={X 1022,Y -651,Z -155,A 0,B -90,C 180,S 6,T 16,E1 0.0,E2 0.0,E3 0.0,E4 0.0,E5 0.0,E6 0.0}
DECL FDAT FP376={TOOL_NO 4,BASE_NO 0,IPO_FRAME #BASE,POINT2[] " "}
DECL LDAT LCPDAT376={VEL 1,ACC 50.000,APO_DIST 500.000,APO_FAC 50.0000,AXIS_VEL 50.000,AXIS_ACC 50.000,ORI_TYP #VAR,CIRC_TYP #BASE,JERK_FAC 50.0000,GEAR_JERK 100.000,EXAX_IGN 0}

DECL E6POS XP377={X 972,Y -651,Z -155,A 0,B -90,C 180,S 6,T 16,E1 0.0,E2 0.0,E3 0.0,E4 0.0,E5 0.0,E6 0.0}
DECL FDAT FP377={TOOL_NO 4,BASE_NO 0,IPO_FRAME #BASE,POINT2[] " "}
DECL LDAT LCPDAT377={VEL 1,ACC 50.000,APO_DIST 500.000,APO_FAC 50.0000,AXIS_VEL 50.000,AXIS_ACC 50.000,ORI_TYP #VAR,CIRC_TYP #BASE,JERK_FAC 50.0000,GEAR_JERK 100.000,EXAX_IGN 0}

DECL E6POS XP378={X 922,Y -651,Z -155,A 0,B -90,C 180,S 6,T 16,E1 0.0,E2 0.0,E3 0.0,E4 0.0,E5 0.0,E6 0.0}
DECL FDAT FP378={TOOL_NO 4,BASE_NO 0,IPO_FRAME #BASE,POINT2[] " "}
DECL LDAT LCPDAT378={VEL 1,ACC 50.000,APO_DIST 500.000,APO_FAC 50.0000,AXIS_VEL 50.000,AXIS_ACC 50.000,ORI_TYP #VAR,CIRC_TYP #BASE,JERK_FAC 50.0000,GEAR_JERK 100.000,EXAX_IGN 0}

DECL E6POS XP379={X 872,Y -651,Z -155,A 0,B -90,C 180,S 6,T 16,E1 0.0,E2 0.0,E3 0.0,E4 0.0,E5 0.0,E6 0.0}
DECL FDAT FP379={TOOL_NO 4,BASE_NO 0,IPO_FRAME #BASE,POINT2[] " "}
DECL LDAT LCPDAT379={VEL 1,ACC 50.000,APO_DIST 500.000,APO_FAC 50.0000,AXIS_VEL 50.000,AXIS_ACC 50.000,ORI_TYP #VAR,CIRC_TYP #BASE,JERK_FAC 50.0000,GEAR_JERK 100.000,EXAX_IGN 0}

DECL E6POS XP380={X 822,Y -651,Z -155,A 0,B -90,C 180,S 6,T 16,E1 0.0,E2 0.0,E3 0.0,E4 0.0,E5 0.0,E6 0.0}
DECL FDAT FP380={TOOL_NO 4,BASE_NO 0,IPO_FRAME #BASE,POINT2[] " "}
DECL LDAT LCPDAT380={VEL 1,ACC 50.000,APO_DIST 500.000,APO_FAC 50.0000,AXIS_VEL 50.000,AXIS_ACC 50.000,ORI_TYP #VAR,CIRC_TYP #BASE,JERK_FAC 50.0000,GEAR_JERK 100.000,EXAX_IGN 0}

DECL E6POS XP381={X 772,Y -651,Z -155,A 0,B -90,C 180,S 6,T 16,E1 0.0,E2 0.0,E3 0.0,E4 0.0,E5 0.0,E6 0.0}
DECL FDAT FP381={TOOL_NO 4,BASE_NO 0,IPO_FRAME #BASE,POINT2[] " "}
DECL LDAT LCPDAT381={VEL 1,ACC 50.000,APO_DIST 500.000,APO_FAC 50.0000,AXIS_VEL 50.000,AXIS_ACC 50.000,ORI_TYP #VAR,CIRC_TYP #BASE,JERK_FAC 50.0000,GEAR_JERK 100.000,EXAX_IGN 0}

DECL E6POS XP382={X 722,Y -651,Z -155,A 0,B -90,C 180,S 6,T 16,E1 0.0,E2 0.0,E3 0.0,E4 0.0,E5 0.0,E6 0.0}
DECL FDAT FP382={TOOL_NO 4,BASE_NO 0,IPO_FRAME #BASE,POINT2[] " "}
DECL LDAT LCPDAT382={VEL 1,ACC 50.000,APO_DIST 500.000,APO_FAC 50.0000,AXIS_VEL 50.000,AXIS_ACC 50.000,ORI_TYP #VAR,CIRC_TYP #BASE,JERK_FAC 50.0000,GEAR_JERK 100.000,EXAX_IGN 0}

DECL E6POS XP383={X 672,Y -651,Z -155,A 0,B -90,C 180,S 6,T 16,E1 0.0,E2 0.0,E3 0.0,E4 0.0,E5 0.0,E6 0.0}
DECL FDAT FP383={TOOL_NO 4,BASE_NO 0,IPO_FRAME #BASE,POINT2[] " "}
DECL LDAT LCPDAT383={VEL 1,ACC 50.000,APO_DIST 500.000,APO_FAC 50.0000,AXIS_VEL 50.000,AXIS_ACC 50.000,ORI_TYP #VAR,CIRC_TYP #BASE,JERK_FAC 50.0000,GEAR_JERK 100.000,EXAX_IGN 0}

DECL E6POS XP384={X 672,Y -651,Z -105,A 0,B -90,C 180,S 6,T 16,E1 0.0,E2 0.0,E3 0.0,E4 0.0,E5 0.0,E6 0.0}
DECL FDAT FP384={TOOL_NO 4,BASE_NO 0,IPO_FRAME #BASE,POINT2[] " "}
DECL LDAT LCPDAT384={VEL 1,ACC 50.000,APO_DIST 500.000,APO_FAC 50.0000,AXIS_VEL 50.000,AXIS_ACC 50.000,ORI_TYP #VAR,CIRC_TYP #BASE,JERK_FAC 50.0000,GEAR_JERK 100.000,EXAX_IGN 0}

DECL E6POS XP385={X 722,Y -651,Z -105,A 0,B -90,C 180,S 6,T 16,E1 0.0,E2 0.0,E3 0.0,E4 0.0,E5 0.0,E6 0.0}
DECL FDAT FP385={TOOL_NO 4,BASE_NO 0,IPO_FRAME #BASE,POINT2[] " "}
DECL LDAT LCPDAT385={VEL 1,ACC 50.000,APO_DIST 500.000,APO_FAC 50.0000,AXIS_VEL 50.000,AXIS_ACC 50.000,ORI_TYP #VAR,CIRC_TYP #BASE,JERK_FAC 50.0000,GEAR_JERK 100.000,EXAX_IGN 0}

DECL E6POS XP386={X 772,Y -651,Z -105,A 0,B -90,C 180,S 6,T 16,E1 0.0,E2 0.0,E3 0.0,E4 0.0,E5 0.0,E6 0.0}
DECL FDAT FP386={TOOL_NO 4,BASE_NO 0,IPO_FRAME #BASE,POINT2[] " "}
DECL LDAT LCPDAT386={VEL 1,ACC 50.000,APO_DIST 500.000,APO_FAC 50.0000,AXIS_VEL 50.000,AXIS_ACC 50.000,ORI_TYP #VAR,CIRC_TYP #BASE,JERK_FAC 50.0000,GEAR_JERK 100.000,EXAX_IGN 0}

DECL E6POS XP387={X 822,Y -651,Z -105,A 0,B -90,C 180,S 6,T 16,E1 0.0,E2 0.0,E3 0.0,E4 0.0,E5 0.0,E6 0.0}
DECL FDAT FP387={TOOL_NO 4,BASE_NO 0,IPO_FRAME #BASE,POINT2[] " "}
DECL LDAT LCPDAT387={VEL 1,ACC 50.000,APO_DIST 500.000,APO_FAC 50.0000,AXIS_VEL 50.000,AXIS_ACC 50.000,ORI_TYP #VAR,CIRC_TYP #BASE,JERK_FAC 50.0000,GEAR_JERK 100.000,EXAX_IGN 0}

DECL E6POS XP388={X 872,Y -651,Z -105,A 0,B -90,C 180,S 6,T 16,E1 0.0,E2 0.0,E3 0.0,E4 0.0,E5 0.0,E6 0.0}
DECL FDAT FP388={TOOL_NO 4,BASE_NO 0,IPO_FRAME #BASE,POINT2[] " "}
DECL LDAT LCPDAT388={VEL 1,ACC 50.000,APO_DIST 500.000,APO_FAC 50.0000,AXIS_VEL 50.000,AXIS_ACC 50.000,ORI_TYP #VAR,CIRC_TYP #BASE,JERK_FAC 50.0000,GEAR_JERK 100.000,EXAX_IGN 0}

DECL E6POS XP389={X 922,Y -651,Z -105,A 0,B -90,C 180,S 6,T 16,E1 0.0,E2 0.0,E3 0.0,E4 0.0,E5 0.0,E6 0.0}
DECL FDAT FP389={TOOL_NO 4,BASE_NO 0,IPO_FRAME #BASE,POINT2[] " "}
DECL LDAT LCPDAT389={VEL 1,ACC 50.000,APO_DIST 500.000,APO_FAC 50.0000,AXIS_VEL 50.000,AXIS_ACC 50.000,ORI_TYP #VAR,CIRC_TYP #BASE,JERK_FAC 50.0000,GEAR_JERK 100.000,EXAX_IGN 0}

DECL E6POS XP390={X 972,Y -651,Z -105,A 0,B -90,C 180,S 6,T 16,E1 0.0,E2 0.0,E3 0.0,E4 0.0,E5 0.0,E6 0.0}
DECL FDAT FP390={TOOL_NO 4,BASE_NO 0,IPO_FRAME #BASE,POINT2[] " "}
DECL LDAT LCPDAT390={VEL 1,ACC 50.000,APO_DIST 500.000,APO_FAC 50.0000,AXIS_VEL 50.000,AXIS_ACC 50.000,ORI_TYP #VAR,CIRC_TYP #BASE,JERK_FAC 50.0000,GEAR_JERK 100.000,EXAX_IGN 0}

DECL E6POS XP391={X 1022,Y -651,Z -105,A 0,B -90,C 180,S 6,T 16,E1 0.0,E2 0.0,E3 0.0,E4 0.0,E5 0.0,E6 0.0}
DECL FDAT FP391={TOOL_NO 4,BASE_NO 0,IPO_FRAME #BASE,POINT2[] " "}
DECL LDAT LCPDAT391={VEL 1,ACC 50.000,APO_DIST 500.000,APO_FAC 50.0000,AXIS_VEL 50.000,AXIS_ACC 50.000,ORI_TYP #VAR,CIRC_TYP #BASE,JERK_FAC 50.0000,GEAR_JERK 100.000,EXAX_IGN 0}

DECL E6POS XP392={X 1072,Y -651,Z -105,A 0,B -90,C 180,S 6,T 16,E1 0.0,E2 0.0,E3 0.0,E4 0.0,E5 0.0,E6 0.0}
DECL FDAT FP392={TOOL_NO 4,BASE_NO 0,IPO_FRAME #BASE,POINT2[] " "}
DECL LDAT LCPDAT392={VEL 1,ACC 50.000,APO_DIST 500.000,APO_FAC 50.0000,AXIS_VEL 50.000,AXIS_ACC 50.000,ORI_TYP #VAR,CIRC_TYP #BASE,JERK_FAC 50.0000,GEAR_JERK 100.000,EXAX_IGN 0}

DECL E6POS XP393={X 1122,Y -651,Z -105,A 0,B -90,C 180,S 6,T 16,E1 0.0,E2 0.0,E3 0.0,E4 0.0,E5 0.0,E6 0.0}
DECL FDAT FP393={TOOL_NO 4,BASE_NO 0,IPO_FRAME #BASE,POINT2[] " "}
DECL LDAT LCPDAT393={VEL 1,ACC 50.000,APO_DIST 500.000,APO_FAC 50.0000,AXIS_VEL 50.000,AXIS_ACC 50.000,ORI_TYP #VAR,CIRC_TYP #BASE,JERK_FAC 50.0000,GEAR_JERK 100.000,EXAX_IGN 0}

DECL E6POS XP394={X 1172,Y -651,Z -105,A 0,B -90,C 180,S 6,T 16,E1 0.0,E2 0.0,E3 0.0,E4 0.0,E5 0.0,E6 0.0}
DECL FDAT FP394={TOOL_NO 4,BASE_NO 0,IPO_FRAME #BASE,POINT2[] " "}
DECL LDAT LCPDAT394={VEL 1,ACC 50.000,APO_DIST 500.000,APO_FAC 50.0000,AXIS_VEL 50.000,AXIS_ACC 50.000,ORI_TYP #VAR,CIRC_TYP #BASE,JERK_FAC 50.0000,GEAR_JERK 100.000,EXAX_IGN 0}

DECL E6POS XP395={X 1222,Y -651,Z -105,A 0,B -90,C 180,S 6,T 16,E1 0.0,E2 0.0,E3 0.0,E4 0.0,E5 0.0,E6 0.0}
DECL FDAT FP395={TOOL_NO 4,BASE_NO 0,IPO_FRAME #BASE,POINT2[] " "}
DECL LDAT LCPDAT395={VEL 1,ACC 50.000,APO_DIST 500.000,APO_FAC 50.0000,AXIS_VEL 50.000,AXIS_ACC 50.000,ORI_TYP #VAR,CIRC_TYP #BASE,JERK_FAC 50.0000,GEAR_JERK 100.000,EXAX_IGN 0}

DECL E6POS XP396={X 1272,Y -651,Z -105,A 0,B -90,C 180,S 6,T 16,E1 0.0,E2 0.0,E3 0.0,E4 0.0,E5 0.0,E6 0.0}
DECL FDAT FP396={TOOL_NO 4,BASE_NO 0,IPO_FRAME #BASE,POINT2[] " "}
DECL LDAT LCPDAT396={VEL 1,ACC 50.000,APO_DIST 500.000,APO_FAC 50.0000,AXIS_VEL 50.000,AXIS_ACC 50.000,ORI_TYP #VAR,CIRC_TYP #BASE,JERK_FAC 50.0000,GEAR_JERK 100.000,EXAX_IGN 0}

DECL E6POS XP397={X 1272,Y -651,Z -55,A 0,B -90,C 180,S 6,T 16,E1 0.0,E2 0.0,E3 0.0,E4 0.0,E5 0.0,E6 0.0}
DECL FDAT FP397={TOOL_NO 4,BASE_NO 0,IPO_FRAME #BASE,POINT2[] " "}
DECL LDAT LCPDAT397={VEL 1,ACC 50.000,APO_DIST 500.000,APO_FAC 50.0000,AXIS_VEL 50.000,AXIS_ACC 50.000,ORI_TYP #VAR,CIRC_TYP #BASE,JERK_FAC 50.0000,GEAR_JERK 100.000,EXAX_IGN 0}

DECL E6POS XP398={X 1222,Y -651,Z -55,A 0,B -90,C 180,S 6,T 16,E1 0.0,E2 0.0,E3 0.0,E4 0.0,E5 0.0,E6 0.0}
DECL FDAT FP398={TOOL_NO 4,BASE_NO 0,IPO_FRAME #BASE,POINT2[] " "}
DECL LDAT LCPDAT398={VEL 1,ACC 50.000,APO_DIST 500.000,APO_FAC 50.0000,AXIS_VEL 50.000,AXIS_ACC 50.000,ORI_TYP #VAR,CIRC_TYP #BASE,JERK_FAC 50.0000,GEAR_JERK 100.000,EXAX_IGN 0}

DECL E6POS XP399={X 1172,Y -651,Z -55,A 0,B -90,C 180,S 6,T 16,E1 0.0,E2 0.0,E3 0.0,E4 0.0,E5 0.0,E6 0.0}
DECL FDAT FP399={TOOL_NO 4,BASE_NO 0,IPO_FRAME #BASE,POINT2[] " "}
DECL LDAT LCPDAT399={VEL 1,ACC 50.000,APO_DIST 500.000,APO_FAC 50.0000,AXIS_VEL 50.000,AXIS_ACC 50.000,ORI_TYP #VAR,CIRC_TYP #BASE,JERK_FAC 50.0000,GEAR_JERK 100.000,EXAX_IGN 0}

DECL E6POS XP400={X 1122,Y -651,Z -55,A 0,B -90,C 180,S 6,T 16,E1 0.0,E2 0.0,E3 0.0,E4 0.0,E5 0.0,E6 0.0}
DECL FDAT FP400={TOOL_NO 4,BASE_NO 0,IPO_FRAME #BASE,POINT2[] " "}
DECL LDAT LCPDAT400={VEL 1,ACC 50.000,APO_DIST 500.000,APO_FAC 50.0000,AXIS_VEL 50.000,AXIS_ACC 50.000,ORI_TYP #VAR,CIRC_TYP #BASE,JERK_FAC 50.0000,GEAR_JERK 100.000,EXAX_IGN 0}

DECL E6POS XP401={X 1072,Y -651,Z -55,A 0,B -90,C 180,S 6,T 16,E1 0.0,E2 0.0,E3 0.0,E4 0.0,E5 0.0,E6 0.0}
DECL FDAT FP401={TOOL_NO 4,BASE_NO 0,IPO_FRAME #BASE,POINT2[] " "}
DECL LDAT LCPDAT401={VEL 1,ACC 50.000,APO_DIST 500.000,APO_FAC 50.0000,AXIS_VEL 50.000,AXIS_ACC 50.000,ORI_TYP #VAR,CIRC_TYP #BASE,JERK_FAC 50.0000,GEAR_JERK 100.000,EXAX_IGN 0}

DECL E6POS XP402={X 1022,Y -651,Z -55,A 0,B -90,C 180,S 6,T 16,E1 0.0,E2 0.0,E3 0.0,E4 0.0,E5 0.0,E6 0.0}
DECL FDAT FP402={TOOL_NO 4,BASE_NO 0,IPO_FRAME #BASE,POINT2[] " "}
DECL LDAT LCPDAT402={VEL 1,ACC 50.000,APO_DIST 500.000,APO_FAC 50.0000,AXIS_VEL 50.000,AXIS_ACC 50.000,ORI_TYP #VAR,CIRC_TYP #BASE,JERK_FAC 50.0000,GEAR_JERK 100.000,EXAX_IGN 0}

DECL E6POS XP403={X 972,Y -651,Z -55,A 0,B -90,C 180,S 6,T 16,E1 0.0,E2 0.0,E3 0.0,E4 0.0,E5 0.0,E6 0.0}
DECL FDAT FP403={TOOL_NO 4,BASE_NO 0,IPO_FRAME #BASE,POINT2[] " "}
DECL LDAT LCPDAT403={VEL 1,ACC 50.000,APO_DIST 500.000,APO_FAC 50.0000,AXIS_VEL 50.000,AXIS_ACC 50.000,ORI_TYP #VAR,CIRC_TYP #BASE,JERK_FAC 50.0000,GEAR_JERK 100.000,EXAX_IGN 0}

DECL E6POS XP404={X 922,Y -651,Z -55,A 0,B -90,C 180,S 6,T 16,E1 0.0,E2 0.0,E3 0.0,E4 0.0,E5 0.0,E6 0.0}
DECL FDAT FP404={TOOL_NO 4,BASE_NO 0,IPO_FRAME #BASE,POINT2[] " "}
DECL LDAT LCPDAT404={VEL 1,ACC 50.000,APO_DIST 500.000,APO_FAC 50.0000,AXIS_VEL 50.000,AXIS_ACC 50.000,ORI_TYP #VAR,CIRC_TYP #BASE,JERK_FAC 50.0000,GEAR_JERK 100.000,EXAX_IGN 0}

DECL E6POS XP405={X 872,Y -651,Z -55,A 0,B -90,C 180,S 6,T 16,E1 0.0,E2 0.0,E3 0.0,E4 0.0,E5 0.0,E6 0.0}
DECL FDAT FP405={TOOL_NO 4,BASE_NO 0,IPO_FRAME #BASE,POINT2[] " "}
DECL LDAT LCPDAT405={VEL 1,ACC 50.000,APO_DIST 500.000,APO_FAC 50.0000,AXIS_VEL 50.000,AXIS_ACC 50.000,ORI_TYP #VAR,CIRC_TYP #BASE,JERK_FAC 50.0000,GEAR_JERK 100.000,EXAX_IGN 0}

DECL E6POS XP406={X 822,Y -651,Z -55,A 0,B -90,C 180,S 6,T 16,E1 0.0,E2 0.0,E3 0.0,E4 0.0,E5 0.0,E6 0.0}
DECL FDAT FP406={TOOL_NO 4,BASE_NO 0,IPO_FRAME #BASE,POINT2[] " "}
DECL LDAT LCPDAT406={VEL 1,ACC 50.000,APO_DIST 500.000,APO_FAC 50.0000,AXIS_VEL 50.000,AXIS_ACC 50.000,ORI_TYP #VAR,CIRC_TYP #BASE,JERK_FAC 50.0000,GEAR_JERK 100.000,EXAX_IGN 0}

DECL E6POS XP407={X 772,Y -651,Z -55,A 0,B -90,C 180,S 6,T 16,E1 0.0,E2 0.0,E3 0.0,E4 0.0,E5 0.0,E6 0.0}
DECL FDAT FP407={TOOL_NO 4,BASE_NO 0,IPO_FRAME #BASE,POINT2[] " "}
DECL LDAT LCPDAT407={VEL 1,ACC 50.000,APO_DIST 500.000,APO_FAC 50.0000,AXIS_VEL 50.000,AXIS_ACC 50.000,ORI_TYP #VAR,CIRC_TYP #BASE,JERK_FAC 50.0000,GEAR_JERK 100.000,EXAX_IGN 0}

DECL E6POS XP408={X 722,Y -651,Z -55,A 0,B -90,C 180,S 6,T 16,E1 0.0,E2 0.0,E3 0.0,E4 0.0,E5 0.0,E6 0.0}
DECL FDAT FP408={TOOL_NO 4,BASE_NO 0,IPO_FRAME #BASE,POINT2[] " "}
DECL LDAT LCPDAT408={VEL 1,ACC 50.000,APO_DIST 500.000,APO_FAC 50.0000,AXIS_VEL 50.000,AXIS_ACC 50.000,ORI_TYP #VAR,CIRC_TYP #BASE,JERK_FAC 50.0000,GEAR_JERK 100.000,EXAX_IGN 0}

DECL E6POS XP409={X 672,Y -651,Z -55,A 0,B -90,C 180,S 6,T 16,E1 0.0,E2 0.0,E3 0.0,E4 0.0,E5 0.0,E6 0.0}
DECL FDAT FP409={TOOL_NO 4,BASE_NO 0,IPO_FRAME #BASE,POINT2[] " "}
DECL LDAT LCPDAT409={VEL 1,ACC 50.000,APO_DIST 500.000,APO_FAC 50.0000,AXIS_VEL 50.000,AXIS_ACC 50.000,ORI_TYP #VAR,CIRC_TYP #BASE,JERK_FAC 50.0000,GEAR_JERK 100.000,EXAX_IGN 0}

DECL E6POS XP410={X 672,Y -651,Z -5,A 0,B -90,C 180,S 6,T 16,E1 0.0,E2 0.0,E3 0.0,E4 0.0,E5 0.0,E6 0.0}
DECL FDAT FP410={TOOL_NO 4,BASE_NO 0,IPO_FRAME #BASE,POINT2[] " "}
DECL LDAT LCPDAT410={VEL 1,ACC 50.000,APO_DIST 500.000,APO_FAC 50.0000,AXIS_VEL 50.000,AXIS_ACC 50.000,ORI_TYP #VAR,CIRC_TYP #BASE,JERK_FAC 50.0000,GEAR_JERK 100.000,EXAX_IGN 0}

DECL E6POS XP411={X 722,Y -651,Z -5,A 0,B -90,C 180,S 6,T 16,E1 0.0,E2 0.0,E3 0.0,E4 0.0,E5 0.0,E6 0.0}
DECL FDAT FP411={TOOL_NO 4,BASE_NO 0,IPO_FRAME #BASE,POINT2[] " "}
DECL LDAT LCPDAT411={VEL 1,ACC 50.000,APO_DIST 500.000,APO_FAC 50.0000,AXIS_VEL 50.000,AXIS_ACC 50.000,ORI_TYP #VAR,CIRC_TYP #BASE,JERK_FAC 50.0000,GEAR_JERK 100.000,EXAX_IGN 0}

DECL E6POS XP412={X 772,Y -651,Z -5,A 0,B -90,C 180,S 6,T 16,E1 0.0,E2 0.0,E3 0.0,E4 0.0,E5 0.0,E6 0.0}
DECL FDAT FP412={TOOL_NO 4,BASE_NO 0,IPO_FRAME #BASE,POINT2[] " "}
DECL LDAT LCPDAT412={VEL 1,ACC 50.000,APO_DIST 500.000,APO_FAC 50.0000,AXIS_VEL 50.000,AXIS_ACC 50.000,ORI_TYP #VAR,CIRC_TYP #BASE,JERK_FAC 50.0000,GEAR_JERK 100.000,EXAX_IGN 0}

DECL E6POS XP413={X 822,Y -651,Z -5,A 0,B -90,C 180,S 6,T 16,E1 0.0,E2 0.0,E3 0.0,E4 0.0,E5 0.0,E6 0.0}
DECL FDAT FP413={TOOL_NO 4,BASE_NO 0,IPO_FRAME #BASE,POINT2[] " "}
DECL LDAT LCPDAT413={VEL 1,ACC 50.000,APO_DIST 500.000,APO_FAC 50.0000,AXIS_VEL 50.000,AXIS_ACC 50.000,ORI_TYP #VAR,CIRC_TYP #BASE,JERK_FAC 50.0000,GEAR_JERK 100.000,EXAX_IGN 0}

DECL E6POS XP414={X 872,Y -651,Z -5,A 0,B -90,C 180,S 6,T 16,E1 0.0,E2 0.0,E3 0.0,E4 0.0,E5 0.0,E6 0.0}
DECL FDAT FP414={TOOL_NO 4,BASE_NO 0,IPO_FRAME #BASE,POINT2[] " "}
DECL LDAT LCPDAT414={VEL 1,ACC 50.000,APO_DIST 500.000,APO_FAC 50.0000,AXIS_VEL 50.000,AXIS_ACC 50.000,ORI_TYP #VAR,CIRC_TYP #BASE,JERK_FAC 50.0000,GEAR_JERK 100.000,EXAX_IGN 0}

DECL E6POS XP415={X 922,Y -651,Z -5,A 0,B -90,C 180,S 6,T 16,E1 0.0,E2 0.0,E3 0.0,E4 0.0,E5 0.0,E6 0.0}
DECL FDAT FP415={TOOL_NO 4,BASE_NO 0,IPO_FRAME #BASE,POINT2[] " "}
DECL LDAT LCPDAT415={VEL 1,ACC 50.000,APO_DIST 500.000,APO_FAC 50.0000,AXIS_VEL 50.000,AXIS_ACC 50.000,ORI_TYP #VAR,CIRC_TYP #BASE,JERK_FAC 50.0000,GEAR_JERK 100.000,EXAX_IGN 0}

DECL E6POS XP416={X 972,Y -651,Z -5,A 0,B -90,C 180,S 6,T 16,E1 0.0,E2 0.0,E3 0.0,E4 0.0,E5 0.0,E6 0.0}
DECL FDAT FP416={TOOL_NO 4,BASE_NO 0,IPO_FRAME #BASE,POINT2[] " "}
DECL LDAT LCPDAT416={VEL 1,ACC 50.000,APO_DIST 500.000,APO_FAC 50.0000,AXIS_VEL 50.000,AXIS_ACC 50.000,ORI_TYP #VAR,CIRC_TYP #BASE,JERK_FAC 50.0000,GEAR_JERK 100.000,EXAX_IGN 0}

DECL E6POS XP417={X 1022,Y -651,Z -5,A 0,B -90,C 180,S 6,T 16,E1 0.0,E2 0.0,E3 0.0,E4 0.0,E5 0.0,E6 0.0}
DECL FDAT FP417={TOOL_NO 4,BASE_NO 0,IPO_FRAME #BASE,POINT2[] " "}
DECL LDAT LCPDAT417={VEL 1,ACC 50.000,APO_DIST 500.000,APO_FAC 50.0000,AXIS_VEL 50.000,AXIS_ACC 50.000,ORI_TYP #VAR,CIRC_TYP #BASE,JERK_FAC 50.0000,GEAR_JERK 100.000,EXAX_IGN 0}

DECL E6POS XP418={X 1072,Y -651,Z -5,A 0,B -90,C 180,S 6,T 16,E1 0.0,E2 0.0,E3 0.0,E4 0.0,E5 0.0,E6 0.0}
DECL FDAT FP418={TOOL_NO 4,BASE_NO 0,IPO_FRAME #BASE,POINT2[] " "}
DECL LDAT LCPDAT418={VEL 1,ACC 50.000,APO_DIST 500.000,APO_FAC 50.0000,AXIS_VEL 50.000,AXIS_ACC 50.000,ORI_TYP #VAR,CIRC_TYP #BASE,JERK_FAC 50.0000,GEAR_JERK 100.000,EXAX_IGN 0}

DECL E6POS XP419={X 1122,Y -651,Z -5,A 0,B -90,C 180,S 6,T 16,E1 0.0,E2 0.0,E3 0.0,E4 0.0,E5 0.0,E6 0.0}
DECL FDAT FP419={TOOL_NO 4,BASE_NO 0,IPO_FRAME #BASE,POINT2[] " "}
DECL LDAT LCPDAT419={VEL 1,ACC 50.000,APO_DIST 500.000,APO_FAC 50.0000,AXIS_VEL 50.000,AXIS_ACC 50.000,ORI_TYP #VAR,CIRC_TYP #BASE,JERK_FAC 50.0000,GEAR_JERK 100.000,EXAX_IGN 0}

DECL E6POS XP420={X 1172,Y -651,Z -5,A 0,B -90,C 180,S 6,T 16,E1 0.0,E2 0.0,E3 0.0,E4 0.0,E5 0.0,E6 0.0}
DECL FDAT FP420={TOOL_NO 4,BASE_NO 0,IPO_FRAME #BASE,POINT2[] " "}
DECL LDAT LCPDAT420={VEL 1,ACC 50.000,APO_DIST 500.000,APO_FAC 50.0000,AXIS_VEL 50.000,AXIS_ACC 50.000,ORI_TYP #VAR,CIRC_TYP #BASE,JERK_FAC 50.0000,GEAR_JERK 100.000,EXAX_IGN 0}

DECL E6POS XP421={X 1222,Y -651,Z -5,A 0,B -90,C 180,S 6,T 16,E1 0.0,E2 0.0,E3 0.0,E4 0.0,E5 0.0,E6 0.0}
DECL FDAT FP421={TOOL_NO 4,BASE_NO 0,IPO_FRAME #BASE,POINT2[] " "}
DECL LDAT LCPDAT421={VEL 1,ACC 50.000,APO_DIST 500.000,APO_FAC 50.0000,AXIS_VEL 50.000,AXIS_ACC 50.000,ORI_TYP #VAR,CIRC_TYP #BASE,JERK_FAC 50.0000,GEAR_JERK 100.000,EXAX_IGN 0}

DECL E6POS XP422={X 1272,Y -651,Z -5,A 0,B -90,C 180,S 6,T 16,E1 0.0,E2 0.0,E3 0.0,E4 0.0,E5 0.0,E6 0.0}
DECL FDAT FP422={TOOL_NO 4,BASE_NO 0,IPO_FRAME #BASE,POINT2[] " "}
DECL LDAT LCPDAT422={VEL 1,ACC 50.000,APO_DIST 500.000,APO_FAC 50.0000,AXIS_VEL 50.000,AXIS_ACC 50.000,ORI_TYP #VAR,CIRC_TYP #BASE,JERK_FAC 50.0000,GEAR_JERK 100.000,EXAX_IGN 0}

DECL E6POS XP423={X 1272,Y -651,Z 45,A 0,B -90,C 180,S 6,T 16,E1 0.0,E2 0.0,E3 0.0,E4 0.0,E5 0.0,E6 0.0}
DECL FDAT FP423={TOOL_NO 4,BASE_NO 0,IPO_FRAME #BASE,POINT2[] " "}
DECL LDAT LCPDAT423={VEL 1,ACC 50.000,APO_DIST 500.000,APO_FAC 50.0000,AXIS_VEL 50.000,AXIS_ACC 50.000,ORI_TYP #VAR,CIRC_TYP #BASE,JERK_FAC 50.0000,GEAR_JERK 100.000,EXAX_IGN 0}

DECL E6POS XP424={X 1222,Y -651,Z 45,A 0,B -90,C 180,S 6,T 16,E1 0.0,E2 0.0,E3 0.0,E4 0.0,E5 0.0,E6 0.0}
DECL FDAT FP424={TOOL_NO 4,BASE_NO 0,IPO_FRAME #BASE,POINT2[] " "}
DECL LDAT LCPDAT424={VEL 1,ACC 50.000,APO_DIST 500.000,APO_FAC 50.0000,AXIS_VEL 50.000,AXIS_ACC 50.000,ORI_TYP #VAR,CIRC_TYP #BASE,JERK_FAC 50.0000,GEAR_JERK 100.000,EXAX_IGN 0}

DECL E6POS XP425={X 1172,Y -651,Z 45,A 0,B -90,C 180,S 6,T 16,E1 0.0,E2 0.0,E3 0.0,E4 0.0,E5 0.0,E6 0.0}
DECL FDAT FP425={TOOL_NO 4,BASE_NO 0,IPO_FRAME #BASE,POINT2[] " "}
DECL LDAT LCPDAT425={VEL 1,ACC 50.000,APO_DIST 500.000,APO_FAC 50.0000,AXIS_VEL 50.000,AXIS_ACC 50.000,ORI_TYP #VAR,CIRC_TYP #BASE,JERK_FAC 50.0000,GEAR_JERK 100.000,EXAX_IGN 0}

DECL E6POS XP426={X 1122,Y -651,Z 45,A 0,B -90,C 180,S 6,T 16,E1 0.0,E2 0.0,E3 0.0,E4 0.0,E5 0.0,E6 0.0}
DECL FDAT FP426={TOOL_NO 4,BASE_NO 0,IPO_FRAME #BASE,POINT2[] " "}
DECL LDAT LCPDAT426={VEL 1,ACC 50.000,APO_DIST 500.000,APO_FAC 50.0000,AXIS_VEL 50.000,AXIS_ACC 50.000,ORI_TYP #VAR,CIRC_TYP #BASE,JERK_FAC 50.0000,GEAR_JERK 100.000,EXAX_IGN 0}

DECL E6POS XP427={X 1072,Y -651,Z 45,A 0,B -90,C 180,S 6,T 16,E1 0.0,E2 0.0,E3 0.0,E4 0.0,E5 0.0,E6 0.0}
DECL FDAT FP427={TOOL_NO 4,BASE_NO 0,IPO_FRAME #BASE,POINT2[] " "}
DECL LDAT LCPDAT427={VEL 1,ACC 50.000,APO_DIST 500.000,APO_FAC 50.0000,AXIS_VEL 50.000,AXIS_ACC 50.000,ORI_TYP #VAR,CIRC_TYP #BASE,JERK_FAC 50.0000,GEAR_JERK 100.000,EXAX_IGN 0}

DECL E6POS XP428={X 1022,Y -651,Z 45,A 0,B -90,C 180,S 6,T 16,E1 0.0,E2 0.0,E3 0.0,E4 0.0,E5 0.0,E6 0.0}
DECL FDAT FP428={TOOL_NO 4,BASE_NO 0,IPO_FRAME #BASE,POINT2[] " "}
DECL LDAT LCPDAT428={VEL 1,ACC 50.000,APO_DIST 500.000,APO_FAC 50.0000,AXIS_VEL 50.000,AXIS_ACC 50.000,ORI_TYP #VAR,CIRC_TYP #BASE,JERK_FAC 50.0000,GEAR_JERK 100.000,EXAX_IGN 0}

DECL E6POS XP429={X 972,Y -651,Z 45,A 0,B -90,C 180,S 6,T 16,E1 0.0,E2 0.0,E3 0.0,E4 0.0,E5 0.0,E6 0.0}
DECL FDAT FP429={TOOL_NO 4,BASE_NO 0,IPO_FRAME #BASE,POINT2[] " "}
DECL LDAT LCPDAT429={VEL 1,ACC 50.000,APO_DIST 500.000,APO_FAC 50.0000,AXIS_VEL 50.000,AXIS_ACC 50.000,ORI_TYP #VAR,CIRC_TYP #BASE,JERK_FAC 50.0000,GEAR_JERK 100.000,EXAX_IGN 0}

DECL E6POS XP430={X 922,Y -651,Z 45,A 0,B -90,C 180,S 6,T 16,E1 0.0,E2 0.0,E3 0.0,E4 0.0,E5 0.0,E6 0.0}
DECL FDAT FP430={TOOL_NO 4,BASE_NO 0,IPO_FRAME #BASE,POINT2[] " "}
DECL LDAT LCPDAT430={VEL 1,ACC 50.000,APO_DIST 500.000,APO_FAC 50.0000,AXIS_VEL 50.000,AXIS_ACC 50.000,ORI_TYP #VAR,CIRC_TYP #BASE,JERK_FAC 50.0000,GEAR_JERK 100.000,EXAX_IGN 0}

DECL E6POS XP431={X 872,Y -651,Z 45,A 0,B -90,C 180,S 6,T 16,E1 0.0,E2 0.0,E3 0.0,E4 0.0,E5 0.0,E6 0.0}
DECL FDAT FP431={TOOL_NO 4,BASE_NO 0,IPO_FRAME #BASE,POINT2[] " "}
DECL LDAT LCPDAT431={VEL 1,ACC 50.000,APO_DIST 500.000,APO_FAC 50.0000,AXIS_VEL 50.000,AXIS_ACC 50.000,ORI_TYP #VAR,CIRC_TYP #BASE,JERK_FAC 50.0000,GEAR_JERK 100.000,EXAX_IGN 0}

DECL E6POS XP432={X 822,Y -651,Z 45,A 0,B -90,C 180,S 6,T 16,E1 0.0,E2 0.0,E3 0.0,E4 0.0,E5 0.0,E6 0.0}
DECL FDAT FP432={TOOL_NO 4,BASE_NO 0,IPO_FRAME #BASE,POINT2[] " "}
DECL LDAT LCPDAT432={VEL 1,ACC 50.000,APO_DIST 500.000,APO_FAC 50.0000,AXIS_VEL 50.000,AXIS_ACC 50.000,ORI_TYP #VAR,CIRC_TYP #BASE,JERK_FAC 50.0000,GEAR_JERK 100.000,EXAX_IGN 0}

DECL E6POS XP433={X 772,Y -651,Z 45,A 0,B -90,C 180,S 6,T 16,E1 0.0,E2 0.0,E3 0.0,E4 0.0,E5 0.0,E6 0.0}
DECL FDAT FP433={TOOL_NO 4,BASE_NO 0,IPO_FRAME #BASE,POINT2[] " "}
DECL LDAT LCPDAT433={VEL 1,ACC 50.000,APO_DIST 500.000,APO_FAC 50.0000,AXIS_VEL 50.000,AXIS_ACC 50.000,ORI_TYP #VAR,CIRC_TYP #BASE,JERK_FAC 50.0000,GEAR_JERK 100.000,EXAX_IGN 0}

DECL E6POS XP434={X 722,Y -651,Z 45,A 0,B -90,C 180,S 6,T 16,E1 0.0,E2 0.0,E3 0.0,E4 0.0,E5 0.0,E6 0.0}
DECL FDAT FP434={TOOL_NO 4,BASE_NO 0,IPO_FRAME #BASE,POINT2[] " "}
DECL LDAT LCPDAT434={VEL 1,ACC 50.000,APO_DIST 500.000,APO_FAC 50.0000,AXIS_VEL 50.000,AXIS_ACC 50.000,ORI_TYP #VAR,CIRC_TYP #BASE,JERK_FAC 50.0000,GEAR_JERK 100.000,EXAX_IGN 0}

DECL E6POS XP435={X 672,Y -651,Z 45,A 0,B -90,C 180,S 6,T 16,E1 0.0,E2 0.0,E3 0.0,E4 0.0,E5 0.0,E6 0.0}
DECL FDAT FP435={TOOL_NO 4,BASE_NO 0,IPO_FRAME #BASE,POINT2[] " "}
DECL LDAT LCPDAT435={VEL 1,ACC 50.000,APO_DIST 500.000,APO_FAC 50.0000,AXIS_VEL 50.000,AXIS_ACC 50.000,ORI_TYP #VAR,CIRC_TYP #BASE,JERK_FAC 50.0000,GEAR_JERK 100.000,EXAX_IGN 0}

DECL E6POS XP436={X 672,Y -651,Z 95,A 0,B -90,C 180,S 6,T 16,E1 0.0,E2 0.0,E3 0.0,E4 0.0,E5 0.0,E6 0.0}
DECL FDAT FP436={TOOL_NO 4,BASE_NO 0,IPO_FRAME #BASE,POINT2[] " "}
DECL LDAT LCPDAT436={VEL 1,ACC 50.000,APO_DIST 500.000,APO_FAC 50.0000,AXIS_VEL 50.000,AXIS_ACC 50.000,ORI_TYP #VAR,CIRC_TYP #BASE,JERK_FAC 50.0000,GEAR_JERK 100.000,EXAX_IGN 0}

DECL E6POS XP437={X 722,Y -651,Z 95,A 0,B -90,C 180,S 6,T 16,E1 0.0,E2 0.0,E3 0.0,E4 0.0,E5 0.0,E6 0.0}
DECL FDAT FP437={TOOL_NO 4,BASE_NO 0,IPO_FRAME #BASE,POINT2[] " "}
DECL LDAT LCPDAT437={VEL 1,ACC 50.000,APO_DIST 500.000,APO_FAC 50.0000,AXIS_VEL 50.000,AXIS_ACC 50.000,ORI_TYP #VAR,CIRC_TYP #BASE,JERK_FAC 50.0000,GEAR_JERK 100.000,EXAX_IGN 0}

DECL E6POS XP438={X 772,Y -651,Z 95,A 0,B -90,C 180,S 6,T 16,E1 0.0,E2 0.0,E3 0.0,E4 0.0,E5 0.0,E6 0.0}
DECL FDAT FP438={TOOL_NO 4,BASE_NO 0,IPO_FRAME #BASE,POINT2[] " "}
DECL LDAT LCPDAT438={VEL 1,ACC 50.000,APO_DIST 500.000,APO_FAC 50.0000,AXIS_VEL 50.000,AXIS_ACC 50.000,ORI_TYP #VAR,CIRC_TYP #BASE,JERK_FAC 50.0000,GEAR_JERK 100.000,EXAX_IGN 0}

DECL E6POS XP439={X 822,Y -651,Z 95,A 0,B -90,C 180,S 6,T 16,E1 0.0,E2 0.0,E3 0.0,E4 0.0,E5 0.0,E6 0.0}
DECL FDAT FP439={TOOL_NO 4,BASE_NO 0,IPO_FRAME #BASE,POINT2[] " "}
DECL LDAT LCPDAT439={VEL 1,ACC 50.000,APO_DIST 500.000,APO_FAC 50.0000,AXIS_VEL 50.000,AXIS_ACC 50.000,ORI_TYP #VAR,CIRC_TYP #BASE,JERK_FAC 50.0000,GEAR_JERK 100.000,EXAX_IGN 0}

DECL E6POS XP440={X 872,Y -651,Z 95,A 0,B -90,C 180,S 6,T 16,E1 0.0,E2 0.0,E3 0.0,E4 0.0,E5 0.0,E6 0.0}
DECL FDAT FP440={TOOL_NO 4,BASE_NO 0,IPO_FRAME #BASE,POINT2[] " "}
DECL LDAT LCPDAT440={VEL 1,ACC 50.000,APO_DIST 500.000,APO_FAC 50.0000,AXIS_VEL 50.000,AXIS_ACC 50.000,ORI_TYP #VAR,CIRC_TYP #BASE,JERK_FAC 50.0000,GEAR_JERK 100.000,EXAX_IGN 0}

DECL E6POS XP441={X 922,Y -651,Z 95,A 0,B -90,C 180,S 6,T 16,E1 0.0,E2 0.0,E3 0.0,E4 0.0,E5 0.0,E6 0.0}
DECL FDAT FP441={TOOL_NO 4,BASE_NO 0,IPO_FRAME #BASE,POINT2[] " "}
DECL LDAT LCPDAT441={VEL 1,ACC 50.000,APO_DIST 500.000,APO_FAC 50.0000,AXIS_VEL 50.000,AXIS_ACC 50.000,ORI_TYP #VAR,CIRC_TYP #BASE,JERK_FAC 50.0000,GEAR_JERK 100.000,EXAX_IGN 0}

DECL E6POS XP442={X 972,Y -651,Z 95,A 0,B -90,C 180,S 6,T 16,E1 0.0,E2 0.0,E3 0.0,E4 0.0,E5 0.0,E6 0.0}
DECL FDAT FP442={TOOL_NO 4,BASE_NO 0,IPO_FRAME #BASE,POINT2[] " "}
DECL LDAT LCPDAT442={VEL 1,ACC 50.000,APO_DIST 500.000,APO_FAC 50.0000,AXIS_VEL 50.000,AXIS_ACC 50.000,ORI_TYP #VAR,CIRC_TYP #BASE,JERK_FAC 50.0000,GEAR_JERK 100.000,EXAX_IGN 0}

DECL E6POS XP443={X 1022,Y -651,Z 95,A 0,B -90,C 180,S 6,T 16,E1 0.0,E2 0.0,E3 0.0,E4 0.0,E5 0.0,E6 0.0}
DECL FDAT FP443={TOOL_NO 4,BASE_NO 0,IPO_FRAME #BASE,POINT2[] " "}
DECL LDAT LCPDAT443={VEL 1,ACC 50.000,APO_DIST 500.000,APO_FAC 50.0000,AXIS_VEL 50.000,AXIS_ACC 50.000,ORI_TYP #VAR,CIRC_TYP #BASE,JERK_FAC 50.0000,GEAR_JERK 100.000,EXAX_IGN 0}

DECL E6POS XP444={X 1072,Y -651,Z 95,A 0,B -90,C 180,S 6,T 16,E1 0.0,E2 0.0,E3 0.0,E4 0.0,E5 0.0,E6 0.0}
DECL FDAT FP444={TOOL_NO 4,BASE_NO 0,IPO_FRAME #BASE,POINT2[] " "}
DECL LDAT LCPDAT444={VEL 1,ACC 50.000,APO_DIST 500.000,APO_FAC 50.0000,AXIS_VEL 50.000,AXIS_ACC 50.000,ORI_TYP #VAR,CIRC_TYP #BASE,JERK_FAC 50.0000,GEAR_JERK 100.000,EXAX_IGN 0}

DECL E6POS XP445={X 1122,Y -651,Z 95,A 0,B -90,C 180,S 6,T 16,E1 0.0,E2 0.0,E3 0.0,E4 0.0,E5 0.0,E6 0.0}
DECL FDAT FP445={TOOL_NO 4,BASE_NO 0,IPO_FRAME #BASE,POINT2[] " "}
DECL LDAT LCPDAT445={VEL 1,ACC 50.000,APO_DIST 500.000,APO_FAC 50.0000,AXIS_VEL 50.000,AXIS_ACC 50.000,ORI_TYP #VAR,CIRC_TYP #BASE,JERK_FAC 50.0000,GEAR_JERK 100.000,EXAX_IGN 0}

DECL E6POS XP446={X 1172,Y -651,Z 95,A 0,B -90,C 180,S 6,T 16,E1 0.0,E2 0.0,E3 0.0,E4 0.0,E5 0.0,E6 0.0}
DECL FDAT FP446={TOOL_NO 4,BASE_NO 0,IPO_FRAME #BASE,POINT2[] " "}
DECL LDAT LCPDAT446={VEL 1,ACC 50.000,APO_DIST 500.000,APO_FAC 50.0000,AXIS_VEL 50.000,AXIS_ACC 50.000,ORI_TYP #VAR,CIRC_TYP #BASE,JERK_FAC 50.0000,GEAR_JERK 100.000,EXAX_IGN 0}

DECL E6POS XP447={X 1222,Y -651,Z 95,A 0,B -90,C 180,S 6,T 16,E1 0.0,E2 0.0,E3 0.0,E4 0.0,E5 0.0,E6 0.0}
DECL FDAT FP447={TOOL_NO 4,BASE_NO 0,IPO_FRAME #BASE,POINT2[] " "}
DECL LDAT LCPDAT447={VEL 1,ACC 50.000,APO_DIST 500.000,APO_FAC 50.0000,AXIS_VEL 50.000,AXIS_ACC 50.000,ORI_TYP #VAR,CIRC_TYP #BASE,JERK_FAC 50.0000,GEAR_JERK 100.000,EXAX_IGN 0}

DECL E6POS XP448={X 1272,Y -651,Z 95,A 0,B -90,C 180,S 6,T 16,E1 0.0,E2 0.0,E3 0.0,E4 0.0,E5 0.0,E6 0.0}
DECL FDAT FP448={TOOL_NO 4,BASE_NO 0,IPO_FRAME #BASE,POINT2[] " "}
DECL LDAT LCPDAT448={VEL 1,ACC 50.000,APO_DIST 500.000,APO_FAC 50.0000,AXIS_VEL 50.000,AXIS_ACC 50.000,ORI_TYP #VAR,CIRC_TYP #BASE,JERK_FAC 50.0000,GEAR_JERK 100.000,EXAX_IGN 0}

DECL E6POS XP449={X 1272,Y -651,Z 145,A 0,B -90,C 180,S 6,T 16,E1 0.0,E2 0.0,E3 0.0,E4 0.0,E5 0.0,E6 0.0}
DECL FDAT FP449={TOOL_NO 4,BASE_NO 0,IPO_FRAME #BASE,POINT2[] " "}
DECL LDAT LCPDAT449={VEL 1,ACC 50.000,APO_DIST 500.000,APO_FAC 50.0000,AXIS_VEL 50.000,AXIS_ACC 50.000,ORI_TYP #VAR,CIRC_TYP #BASE,JERK_FAC 50.0000,GEAR_JERK 100.000,EXAX_IGN 0}

DECL E6POS XP450={X 1222,Y -651,Z 145,A 0,B -90,C 180,S 6,T 16,E1 0.0,E2 0.0,E3 0.0,E4 0.0,E5 0.0,E6 0.0}
DECL FDAT FP450={TOOL_NO 4,BASE_NO 0,IPO_FRAME #BASE,POINT2[] " "}
DECL LDAT LCPDAT450={VEL 1,ACC 50.000,APO_DIST 500.000,APO_FAC 50.0000,AXIS_VEL 50.000,AXIS_ACC 50.000,ORI_TYP #VAR,CIRC_TYP #BASE,JERK_FAC 50.0000,GEAR_JERK 100.000,EXAX_IGN 0}

DECL E6POS XP451={X 1172,Y -651,Z 145,A 0,B -90,C 180,S 6,T 16,E1 0.0,E2 0.0,E3 0.0,E4 0.0,E5 0.0,E6 0.0}
DECL FDAT FP451={TOOL_NO 4,BASE_NO 0,IPO_FRAME #BASE,POINT2[] " "}
DECL LDAT LCPDAT451={VEL 1,ACC 50.000,APO_DIST 500.000,APO_FAC 50.0000,AXIS_VEL 50.000,AXIS_ACC 50.000,ORI_TYP #VAR,CIRC_TYP #BASE,JERK_FAC 50.0000,GEAR_JERK 100.000,EXAX_IGN 0}

DECL E6POS XP452={X 1122,Y -651,Z 145,A 0,B -90,C 180,S 6,T 16,E1 0.0,E2 0.0,E3 0.0,E4 0.0,E5 0.0,E6 0.0}
DECL FDAT FP452={TOOL_NO 4,BASE_NO 0,IPO_FRAME #BASE,POINT2[] " "}
DECL LDAT LCPDAT452={VEL 1,ACC 50.000,APO_DIST 500.000,APO_FAC 50.0000,AXIS_VEL 50.000,AXIS_ACC 50.000,ORI_TYP #VAR,CIRC_TYP #BASE,JERK_FAC 50.0000,GEAR_JERK 100.000,EXAX_IGN 0}

DECL E6POS XP453={X 1072,Y -651,Z 145,A 0,B -90,C 180,S 6,T 16,E1 0.0,E2 0.0,E3 0.0,E4 0.0,E5 0.0,E6 0.0}
DECL FDAT FP453={TOOL_NO 4,BASE_NO 0,IPO_FRAME #BASE,POINT2[] " "}
DECL LDAT LCPDAT453={VEL 1,ACC 50.000,APO_DIST 500.000,APO_FAC 50.0000,AXIS_VEL 50.000,AXIS_ACC 50.000,ORI_TYP #VAR,CIRC_TYP #BASE,JERK_FAC 50.0000,GEAR_JERK 100.000,EXAX_IGN 0}

DECL E6POS XP454={X 1022,Y -651,Z 145,A 0,B -90,C 180,S 6,T 16,E1 0.0,E2 0.0,E3 0.0,E4 0.0,E5 0.0,E6 0.0}
DECL FDAT FP454={TOOL_NO 4,BASE_NO 0,IPO_FRAME #BASE,POINT2[] " "}
DECL LDAT LCPDAT454={VEL 1,ACC 50.000,APO_DIST 500.000,APO_FAC 50.0000,AXIS_VEL 50.000,AXIS_ACC 50.000,ORI_TYP #VAR,CIRC_TYP #BASE,JERK_FAC 50.0000,GEAR_JERK 100.000,EXAX_IGN 0}

DECL E6POS XP455={X 972,Y -651,Z 145,A 0,B -90,C 180,S 6,T 16,E1 0.0,E2 0.0,E3 0.0,E4 0.0,E5 0.0,E6 0.0}
DECL FDAT FP455={TOOL_NO 4,BASE_NO 0,IPO_FRAME #BASE,POINT2[] " "}
DECL LDAT LCPDAT455={VEL 1,ACC 50.000,APO_DIST 500.000,APO_FAC 50.0000,AXIS_VEL 50.000,AXIS_ACC 50.000,ORI_TYP #VAR,CIRC_TYP #BASE,JERK_FAC 50.0000,GEAR_JERK 100.000,EXAX_IGN 0}

DECL E6POS XP456={X 922,Y -651,Z 145,A 0,B -90,C 180,S 6,T 16,E1 0.0,E2 0.0,E3 0.0,E4 0.0,E5 0.0,E6 0.0}
DECL FDAT FP456={TOOL_NO 4,BASE_NO 0,IPO_FRAME #BASE,POINT2[] " "}
DECL LDAT LCPDAT456={VEL 1,ACC 50.000,APO_DIST 500.000,APO_FAC 50.0000,AXIS_VEL 50.000,AXIS_ACC 50.000,ORI_TYP #VAR,CIRC_TYP #BASE,JERK_FAC 50.0000,GEAR_JERK 100.000,EXAX_IGN 0}

DECL E6POS XP457={X 872,Y -651,Z 145,A 0,B -90,C 180,S 6,T 16,E1 0.0,E2 0.0,E3 0.0,E4 0.0,E5 0.0,E6 0.0}
DECL FDAT FP457={TOOL_NO 4,BASE_NO 0,IPO_FRAME #BASE,POINT2[] " "}
DECL LDAT LCPDAT457={VEL 1,ACC 50.000,APO_DIST 500.000,APO_FAC 50.0000,AXIS_VEL 50.000,AXIS_ACC 50.000,ORI_TYP #VAR,CIRC_TYP #BASE,JERK_FAC 50.0000,GEAR_JERK 100.000,EXAX_IGN 0}

DECL E6POS XP458={X 822,Y -651,Z 145,A 0,B -90,C 180,S 6,T 16,E1 0.0,E2 0.0,E3 0.0,E4 0.0,E5 0.0,E6 0.0}
DECL FDAT FP458={TOOL_NO 4,BASE_NO 0,IPO_FRAME #BASE,POINT2[] " "}
DECL LDAT LCPDAT458={VEL 1,ACC 50.000,APO_DIST 500.000,APO_FAC 50.0000,AXIS_VEL 50.000,AXIS_ACC 50.000,ORI_TYP #VAR,CIRC_TYP #BASE,JERK_FAC 50.0000,GEAR_JERK 100.000,EXAX_IGN 0}

DECL E6POS XP459={X 772,Y -651,Z 145,A 0,B -90,C 180,S 6,T 16,E1 0.0,E2 0.0,E3 0.0,E4 0.0,E5 0.0,E6 0.0}
DECL FDAT FP459={TOOL_NO 4,BASE_NO 0,IPO_FRAME #BASE,POINT2[] " "}
DECL LDAT LCPDAT459={VEL 1,ACC 50.000,APO_DIST 500.000,APO_FAC 50.0000,AXIS_VEL 50.000,AXIS_ACC 50.000,ORI_TYP #VAR,CIRC_TYP #BASE,JERK_FAC 50.0000,GEAR_JERK 100.000,EXAX_IGN 0}

DECL E6POS XP460={X 722,Y -651,Z 145,A 0,B -90,C 180,S 6,T 16,E1 0.0,E2 0.0,E3 0.0,E4 0.0,E5 0.0,E6 0.0}
DECL FDAT FP460={TOOL_NO 4,BASE_NO 0,IPO_FRAME #BASE,POINT2[] " "}
DECL LDAT LCPDAT460={VEL 1,ACC 50.000,APO_DIST 500.000,APO_FAC 50.0000,AXIS_VEL 50.000,AXIS_ACC 50.000,ORI_TYP #VAR,CIRC_TYP #BASE,JERK_FAC 50.0000,GEAR_JERK 100.000,EXAX_IGN 0}

DECL E6POS XP461={X 672,Y -651,Z 145,A 0,B -90,C 180,S 6,T 16,E1 0.0,E2 0.0,E3 0.0,E4 0.0,E5 0.0,E6 0.0}
DECL FDAT FP461={TOOL_NO 4,BASE_NO 0,IPO_FRAME #BASE,POINT2[] " "}
DECL LDAT LCPDAT461={VEL 1,ACC 50.000,APO_DIST 500.000,APO_FAC 50.0000,AXIS_VEL 50.000,AXIS_ACC 50.000,ORI_TYP #VAR,CIRC_TYP #BASE,JERK_FAC 50.0000,GEAR_JERK 100.000,EXAX_IGN 0}

DECL E6POS XP462={X 672,Y -651,Z 195,A 0,B -90,C 180,S 6,T 16,E1 0.0,E2 0.0,E3 0.0,E4 0.0,E5 0.0,E6 0.0}
DECL FDAT FP462={TOOL_NO 4,BASE_NO 0,IPO_FRAME #BASE,POINT2[] " "}
DECL LDAT LCPDAT462={VEL 1,ACC 50.000,APO_DIST 500.000,APO_FAC 50.0000,AXIS_VEL 50.000,AXIS_ACC 50.000,ORI_TYP #VAR,CIRC_TYP #BASE,JERK_FAC 50.0000,GEAR_JERK 100.000,EXAX_IGN 0}

DECL E6POS XP463={X 722,Y -651,Z 195,A 0,B -90,C 180,S 6,T 16,E1 0.0,E2 0.0,E3 0.0,E4 0.0,E5 0.0,E6 0.0}
DECL FDAT FP463={TOOL_NO 4,BASE_NO 0,IPO_FRAME #BASE,POINT2[] " "}
DECL LDAT LCPDAT463={VEL 1,ACC 50.000,APO_DIST 500.000,APO_FAC 50.0000,AXIS_VEL 50.000,AXIS_ACC 50.000,ORI_TYP #VAR,CIRC_TYP #BASE,JERK_FAC 50.0000,GEAR_JERK 100.000,EXAX_IGN 0}

DECL E6POS XP464={X 772,Y -651,Z 195,A 0,B -90,C 180,S 6,T 16,E1 0.0,E2 0.0,E3 0.0,E4 0.0,E5 0.0,E6 0.0}
DECL FDAT FP464={TOOL_NO 4,BASE_NO 0,IPO_FRAME #BASE,POINT2[] " "}
DECL LDAT LCPDAT464={VEL 1,ACC 50.000,APO_DIST 500.000,APO_FAC 50.0000,AXIS_VEL 50.000,AXIS_ACC 50.000,ORI_TYP #VAR,CIRC_TYP #BASE,JERK_FAC 50.0000,GEAR_JERK 100.000,EXAX_IGN 0}

DECL E6POS XP465={X 822,Y -651,Z 195,A 0,B -90,C 180,S 6,T 16,E1 0.0,E2 0.0,E3 0.0,E4 0.0,E5 0.0,E6 0.0}
DECL FDAT FP465={TOOL_NO 4,BASE_NO 0,IPO_FRAME #BASE,POINT2[] " "}
DECL LDAT LCPDAT465={VEL 1,ACC 50.000,APO_DIST 500.000,APO_FAC 50.0000,AXIS_VEL 50.000,AXIS_ACC 50.000,ORI_TYP #VAR,CIRC_TYP #BASE,JERK_FAC 50.0000,GEAR_JERK 100.000,EXAX_IGN 0}

DECL E6POS XP466={X 872,Y -651,Z 195,A 0,B -90,C 180,S 6,T 16,E1 0.0,E2 0.0,E3 0.0,E4 0.0,E5 0.0,E6 0.0}
DECL FDAT FP466={TOOL_NO 4,BASE_NO 0,IPO_FRAME #BASE,POINT2[] " "}
DECL LDAT LCPDAT466={VEL 1,ACC 50.000,APO_DIST 500.000,APO_FAC 50.0000,AXIS_VEL 50.000,AXIS_ACC 50.000,ORI_TYP #VAR,CIRC_TYP #BASE,JERK_FAC 50.0000,GEAR_JERK 100.000,EXAX_IGN 0}

DECL E6POS XP467={X 922,Y -651,Z 195,A 0,B -90,C 180,S 6,T 16,E1 0.0,E2 0.0,E3 0.0,E4 0.0,E5 0.0,E6 0.0}
DECL FDAT FP467={TOOL_NO 4,BASE_NO 0,IPO_FRAME #BASE,POINT2[] " "}
DECL LDAT LCPDAT467={VEL 1,ACC 50.000,APO_DIST 500.000,APO_FAC 50.0000,AXIS_VEL 50.000,AXIS_ACC 50.000,ORI_TYP #VAR,CIRC_TYP #BASE,JERK_FAC 50.0000,GEAR_JERK 100.000,EXAX_IGN 0}

DECL E6POS XP468={X 972,Y -651,Z 195,A 0,B -90,C 180,S 6,T 16,E1 0.0,E2 0.0,E3 0.0,E4 0.0,E5 0.0,E6 0.0}
DECL FDAT FP468={TOOL_NO 4,BASE_NO 0,IPO_FRAME #BASE,POINT2[] " "}
DECL LDAT LCPDAT468={VEL 1,ACC 50.000,APO_DIST 500.000,APO_FAC 50.0000,AXIS_VEL 50.000,AXIS_ACC 50.000,ORI_TYP #VAR,CIRC_TYP #BASE,JERK_FAC 50.0000,GEAR_JERK 100.000,EXAX_IGN 0}

DECL E6POS XP469={X 1022,Y -651,Z 195,A 0,B -90,C 180,S 6,T 16,E1 0.0,E2 0.0,E3 0.0,E4 0.0,E5 0.0,E6 0.0}
DECL FDAT FP469={TOOL_NO 4,BASE_NO 0,IPO_FRAME #BASE,POINT2[] " "}
DECL LDAT LCPDAT469={VEL 1,ACC 50.000,APO_DIST 500.000,APO_FAC 50.0000,AXIS_VEL 50.000,AXIS_ACC 50.000,ORI_TYP #VAR,CIRC_TYP #BASE,JERK_FAC 50.0000,GEAR_JERK 100.000,EXAX_IGN 0}

DECL E6POS XP470={X 1072,Y -651,Z 195,A 0,B -90,C 180,S 6,T 16,E1 0.0,E2 0.0,E3 0.0,E4 0.0,E5 0.0,E6 0.0}
DECL FDAT FP470={TOOL_NO 4,BASE_NO 0,IPO_FRAME #BASE,POINT2[] " "}
DECL LDAT LCPDAT470={VEL 1,ACC 50.000,APO_DIST 500.000,APO_FAC 50.0000,AXIS_VEL 50.000,AXIS_ACC 50.000,ORI_TYP #VAR,CIRC_TYP #BASE,JERK_FAC 50.0000,GEAR_JERK 100.000,EXAX_IGN 0}

DECL E6POS XP471={X 1122,Y -651,Z 195,A 0,B -90,C 180,S 6,T 16,E1 0.0,E2 0.0,E3 0.0,E4 0.0,E5 0.0,E6 0.0}
DECL FDAT FP471={TOOL_NO 4,BASE_NO 0,IPO_FRAME #BASE,POINT2[] " "}
DECL LDAT LCPDAT471={VEL 1,ACC 50.000,APO_DIST 500.000,APO_FAC 50.0000,AXIS_VEL 50.000,AXIS_ACC 50.000,ORI_TYP #VAR,CIRC_TYP #BASE,JERK_FAC 50.0000,GEAR_JERK 100.000,EXAX_IGN 0}

DECL E6POS XP472={X 1172,Y -651,Z 195,A 0,B -90,C 180,S 6,T 16,E1 0.0,E2 0.0,E3 0.0,E4 0.0,E5 0.0,E6 0.0}
DECL FDAT FP472={TOOL_NO 4,BASE_NO 0,IPO_FRAME #BASE,POINT2[] " "}
DECL LDAT LCPDAT472={VEL 1,ACC 50.000,APO_DIST 500.000,APO_FAC 50.0000,AXIS_VEL 50.000,AXIS_ACC 50.000,ORI_TYP #VAR,CIRC_TYP #BASE,JERK_FAC 50.0000,GEAR_JERK 100.000,EXAX_IGN 0}

DECL E6POS XP473={X 1222,Y -651,Z 195,A 0,B -90,C 180,S 6,T 16,E1 0.0,E2 0.0,E3 0.0,E4 0.0,E5 0.0,E6 0.0}
DECL FDAT FP473={TOOL_NO 4,BASE_NO 0,IPO_FRAME #BASE,POINT2[] " "}
DECL LDAT LCPDAT473={VEL 1,ACC 50.000,APO_DIST 500.000,APO_FAC 50.0000,AXIS_VEL 50.000,AXIS_ACC 50.000,ORI_TYP #VAR,CIRC_TYP #BASE,JERK_FAC 50.0000,GEAR_JERK 100.000,EXAX_IGN 0}

DECL E6POS XP474={X 1272,Y -651,Z 195,A 0,B -90,C 180,S 6,T 16,E1 0.0,E2 0.0,E3 0.0,E4 0.0,E5 0.0,E6 0.0}
DECL FDAT FP474={TOOL_NO 4,BASE_NO 0,IPO_FRAME #BASE,POINT2[] " "}
DECL LDAT LCPDAT474={VEL 1,ACC 50.000,APO_DIST 500.000,APO_FAC 50.0000,AXIS_VEL 50.000,AXIS_ACC 50.000,ORI_TYP #VAR,CIRC_TYP #BASE,JERK_FAC 50.0000,GEAR_JERK 100.000,EXAX_IGN 0}

DECL E6POS XP475={X 1272,Y -651,Z 245,A 0,B -90,C 180,S 6,T 16,E1 0.0,E2 0.0,E3 0.0,E4 0.0,E5 0.0,E6 0.0}
DECL FDAT FP475={TOOL_NO 4,BASE_NO 0,IPO_FRAME #BASE,POINT2[] " "}
DECL LDAT LCPDAT475={VEL 1,ACC 50.000,APO_DIST 500.000,APO_FAC 50.0000,AXIS_VEL 50.000,AXIS_ACC 50.000,ORI_TYP #VAR,CIRC_TYP #BASE,JERK_FAC 50.0000,GEAR_JERK 100.000,EXAX_IGN 0}

DECL E6POS XP476={X 1222,Y -651,Z 245,A 0,B -90,C 180,S 6,T 16,E1 0.0,E2 0.0,E3 0.0,E4 0.0,E5 0.0,E6 0.0}
DECL FDAT FP476={TOOL_NO 4,BASE_NO 0,IPO_FRAME #BASE,POINT2[] " "}
DECL LDAT LCPDAT476={VEL 1,ACC 50.000,APO_DIST 500.000,APO_FAC 50.0000,AXIS_VEL 50.000,AXIS_ACC 50.000,ORI_TYP #VAR,CIRC_TYP #BASE,JERK_FAC 50.0000,GEAR_JERK 100.000,EXAX_IGN 0}

DECL E6POS XP477={X 1172,Y -651,Z 245,A 0,B -90,C 180,S 6,T 16,E1 0.0,E2 0.0,E3 0.0,E4 0.0,E5 0.0,E6 0.0}
DECL FDAT FP477={TOOL_NO 4,BASE_NO 0,IPO_FRAME #BASE,POINT2[] " "}
DECL LDAT LCPDAT477={VEL 1,ACC 50.000,APO_DIST 500.000,APO_FAC 50.0000,AXIS_VEL 50.000,AXIS_ACC 50.000,ORI_TYP #VAR,CIRC_TYP #BASE,JERK_FAC 50.0000,GEAR_JERK 100.000,EXAX_IGN 0}

DECL E6POS XP478={X 1122,Y -651,Z 245,A 0,B -90,C 180,S 6,T 16,E1 0.0,E2 0.0,E3 0.0,E4 0.0,E5 0.0,E6 0.0}
DECL FDAT FP478={TOOL_NO 4,BASE_NO 0,IPO_FRAME #BASE,POINT2[] " "}
DECL LDAT LCPDAT478={VEL 1,ACC 50.000,APO_DIST 500.000,APO_FAC 50.0000,AXIS_VEL 50.000,AXIS_ACC 50.000,ORI_TYP #VAR,CIRC_TYP #BASE,JERK_FAC 50.0000,GEAR_JERK 100.000,EXAX_IGN 0}

DECL E6POS XP479={X 1072,Y -651,Z 245,A 0,B -90,C 180,S 6,T 16,E1 0.0,E2 0.0,E3 0.0,E4 0.0,E5 0.0,E6 0.0}
DECL FDAT FP479={TOOL_NO 4,BASE_NO 0,IPO_FRAME #BASE,POINT2[] " "}
DECL LDAT LCPDAT479={VEL 1,ACC 50.000,APO_DIST 500.000,APO_FAC 50.0000,AXIS_VEL 50.000,AXIS_ACC 50.000,ORI_TYP #VAR,CIRC_TYP #BASE,JERK_FAC 50.0000,GEAR_JERK 100.000,EXAX_IGN 0}

DECL E6POS XP480={X 1022,Y -651,Z 245,A 0,B -90,C 180,S 6,T 16,E1 0.0,E2 0.0,E3 0.0,E4 0.0,E5 0.0,E6 0.0}
DECL FDAT FP480={TOOL_NO 4,BASE_NO 0,IPO_FRAME #BASE,POINT2[] " "}
DECL LDAT LCPDAT480={VEL 1,ACC 50.000,APO_DIST 500.000,APO_FAC 50.0000,AXIS_VEL 50.000,AXIS_ACC 50.000,ORI_TYP #VAR,CIRC_TYP #BASE,JERK_FAC 50.0000,GEAR_JERK 100.000,EXAX_IGN 0}

DECL E6POS XP481={X 972,Y -651,Z 245,A 0,B -90,C 180,S 6,T 16,E1 0.0,E2 0.0,E3 0.0,E4 0.0,E5 0.0,E6 0.0}
DECL FDAT FP481={TOOL_NO 4,BASE_NO 0,IPO_FRAME #BASE,POINT2[] " "}
DECL LDAT LCPDAT481={VEL 1,ACC 50.000,APO_DIST 500.000,APO_FAC 50.0000,AXIS_VEL 50.000,AXIS_ACC 50.000,ORI_TYP #VAR,CIRC_TYP #BASE,JERK_FAC 50.0000,GEAR_JERK 100.000,EXAX_IGN 0}

DECL E6POS XP482={X 922,Y -651,Z 245,A 0,B -90,C 180,S 6,T 16,E1 0.0,E2 0.0,E3 0.0,E4 0.0,E5 0.0,E6 0.0}
DECL FDAT FP482={TOOL_NO 4,BASE_NO 0,IPO_FRAME #BASE,POINT2[] " "}
DECL LDAT LCPDAT482={VEL 1,ACC 50.000,APO_DIST 500.000,APO_FAC 50.0000,AXIS_VEL 50.000,AXIS_ACC 50.000,ORI_TYP #VAR,CIRC_TYP #BASE,JERK_FAC 50.0000,GEAR_JERK 100.000,EXAX_IGN 0}

DECL E6POS XP483={X 872,Y -651,Z 245,A 0,B -90,C 180,S 6,T 16,E1 0.0,E2 0.0,E3 0.0,E4 0.0,E5 0.0,E6 0.0}
DECL FDAT FP483={TOOL_NO 4,BASE_NO 0,IPO_FRAME #BASE,POINT2[] " "}
DECL LDAT LCPDAT483={VEL 1,ACC 50.000,APO_DIST 500.000,APO_FAC 50.0000,AXIS_VEL 50.000,AXIS_ACC 50.000,ORI_TYP #VAR,CIRC_TYP #BASE,JERK_FAC 50.0000,GEAR_JERK 100.000,EXAX_IGN 0}

DECL E6POS XP484={X 822,Y -651,Z 245,A 0,B -90,C 180,S 6,T 16,E1 0.0,E2 0.0,E3 0.0,E4 0.0,E5 0.0,E6 0.0}
DECL FDAT FP484={TOOL_NO 4,BASE_NO 0,IPO_FRAME #BASE,POINT2[] " "}
DECL LDAT LCPDAT484={VEL 1,ACC 50.000,APO_DIST 500.000,APO_FAC 50.0000,AXIS_VEL 50.000,AXIS_ACC 50.000,ORI_TYP #VAR,CIRC_TYP #BASE,JERK_FAC 50.0000,GEAR_JERK 100.000,EXAX_IGN 0}

DECL E6POS XP485={X 772,Y -651,Z 245,A 0,B -90,C 180,S 6,T 16,E1 0.0,E2 0.0,E3 0.0,E4 0.0,E5 0.0,E6 0.0}
DECL FDAT FP485={TOOL_NO 4,BASE_NO 0,IPO_FRAME #BASE,POINT2[] " "}
DECL LDAT LCPDAT485={VEL 1,ACC 50.000,APO_DIST 500.000,APO_FAC 50.0000,AXIS_VEL 50.000,AXIS_ACC 50.000,ORI_TYP #VAR,CIRC_TYP #BASE,JERK_FAC 50.0000,GEAR_JERK 100.000,EXAX_IGN 0}

DECL E6POS XP486={X 722,Y -651,Z 245,A 0,B -90,C 180,S 6,T 16,E1 0.0,E2 0.0,E3 0.0,E4 0.0,E5 0.0,E6 0.0}
DECL FDAT FP486={TOOL_NO 4,BASE_NO 0,IPO_FRAME #BASE,POINT2[] " "}
DECL LDAT LCPDAT486={VEL 1,ACC 50.000,APO_DIST 500.000,APO_FAC 50.0000,AXIS_VEL 50.000,AXIS_ACC 50.000,ORI_TYP #VAR,CIRC_TYP #BASE,JERK_FAC 50.0000,GEAR_JERK 100.000,EXAX_IGN 0}

DECL E6POS XP487={X 672,Y -651,Z 245,A 0,B -90,C 180,S 6,T 16,E1 0.0,E2 0.0,E3 0.0,E4 0.0,E5 0.0,E6 0.0}
DECL FDAT FP487={TOOL_NO 4,BASE_NO 0,IPO_FRAME #BASE,POINT2[] " "}
DECL LDAT LCPDAT487={VEL 1,ACC 50.000,APO_DIST 500.000,APO_FAC 50.0000,AXIS_VEL 50.000,AXIS_ACC 50.000,ORI_TYP #VAR,CIRC_TYP #BASE,JERK_FAC 50.0000,GEAR_JERK 100.000,EXAX_IGN 0}

DECL E6POS XP488={X 1272,Y -651,Z 445,A 0,B -90,C 180,S 6,T 16,E1 0.0,E2 0.0,E3 0.0,E4 0.0,E5 0.0,E6 0.0}
DECL FDAT FP488={TOOL_NO 4,BASE_NO 0,IPO_FRAME #BASE,POINT2[] " "}
DECL LDAT LCPDAT488={VEL 0.25,ACC 12.000,APO_DIST 500.000,APO_FAC 50.0000,AXIS_VEL 12.000,AXIS_ACC 12.000,ORI_TYP #VAR,CIRC_TYP #BASE,JERK_FAC 50.0000,GEAR_JERK 100.000,EXAX_IGN 0}

DECL E6POS XP489={X 1272,Y -51,Z 445,A 0,B -90,C 180,S 6,T 50,E1 0.0,E2 0.0,E3 0.0,E4 0.0,E5 0.0,E6 0.0}
DECL FDAT FP489={TOOL_NO 4,BASE_NO 0,IPO_FRAME #BASE,POINT2[] " "}
DECL PDAT PPDAT489={VEL 20.000,ACC 20.000,APO_DIST 500.000,APO_MODE #CDIS,GEAR_JERK 100.000,EXAX_IGN 0}

DECL E6POS XP490={X 1272,Y 549,Z 445,A 0,B -90,C 180,S 6,T 16,E1 0.0,E2 0.0,E3 0.0,E4 0.0,E5 0.0,E6 0.0}
DECL FDAT FP490={TOOL_NO 4,BASE_NO 0,IPO_FRAME #BASE,POINT2[] " "}
DECL LDAT LCPDAT490={VEL 0.25,ACC 12.000,APO_DIST 500.000,APO_FAC 50.0000,AXIS_VEL 12.000,AXIS_ACC 12.000,ORI_TYP #VAR,CIRC_TYP #BASE,JERK_FAC 50.0000,GEAR_JERK 100.000,EXAX_IGN 0}

DECL E6POS XP491={X 1272,Y 549,Z -355,A 0,B -90,C 180,S 6,T 16,E1 0.0,E2 0.0,E3 0.0,E4 0.0,E5 0.0,E6 0.0}
DECL FDAT FP491={TOOL_NO 4,BASE_NO 0,IPO_FRAME #BASE,POINT2[] " "}
DECL LDAT LCPDAT491={VEL 1,ACC 50.000,APO_DIST 500.000,APO_FAC 50.0000,AXIS_VEL 50.000,AXIS_ACC 50.000,ORI_TYP #VAR,CIRC_TYP #BASE,JERK_FAC 50.0000,GEAR_JERK 100.000,EXAX_IGN 0}

DECL E6POS XP492={X 1222,Y 549,Z -355,A 0,B -90,C 180,S 6,T 16,E1 0.0,E2 0.0,E3 0.0,E4 0.0,E5 0.0,E6 0.0}
DECL FDAT FP492={TOOL_NO 4,BASE_NO 0,IPO_FRAME #BASE,POINT2[] " "}
DECL LDAT LCPDAT492={VEL 1,ACC 50.000,APO_DIST 500.000,APO_FAC 50.0000,AXIS_VEL 50.000,AXIS_ACC 50.000,ORI_TYP #VAR,CIRC_TYP #BASE,JERK_FAC 50.0000,GEAR_JERK 100.000,EXAX_IGN 0}

DECL E6POS XP493={X 1172,Y 549,Z -355,A 0,B -90,C 180,S 6,T 16,E1 0.0,E2 0.0,E3 0.0,E4 0.0,E5 0.0,E6 0.0}
DECL FDAT FP493={TOOL_NO 4,BASE_NO 0,IPO_FRAME #BASE,POINT2[] " "}
DECL LDAT LCPDAT493={VEL 1,ACC 50.000,APO_DIST 500.000,APO_FAC 50.0000,AXIS_VEL 50.000,AXIS_ACC 50.000,ORI_TYP #VAR,CIRC_TYP #BASE,JERK_FAC 50.0000,GEAR_JERK 100.000,EXAX_IGN 0}

DECL E6POS XP494={X 1122,Y 549,Z -355,A 0,B -90,C 180,S 6,T 16,E1 0.0,E2 0.0,E3 0.0,E4 0.0,E5 0.0,E6 0.0}
DECL FDAT FP494={TOOL_NO 4,BASE_NO 0,IPO_FRAME #BASE,POINT2[] " "}
DECL LDAT LCPDAT494={VEL 1,ACC 50.000,APO_DIST 500.000,APO_FAC 50.0000,AXIS_VEL 50.000,AXIS_ACC 50.000,ORI_TYP #VAR,CIRC_TYP #BASE,JERK_FAC 50.0000,GEAR_JERK 100.000,EXAX_IGN 0}

DECL E6POS XP495={X 1072,Y 549,Z -355,A 0,B -90,C 180,S 6,T 16,E1 0.0,E2 0.0,E3 0.0,E4 0.0,E5 0.0,E6 0.0}
DECL FDAT FP495={TOOL_NO 4,BASE_NO 0,IPO_FRAME #BASE,POINT2[] " "}
DECL LDAT LCPDAT495={VEL 1,ACC 50.000,APO_DIST 500.000,APO_FAC 50.0000,AXIS_VEL 50.000,AXIS_ACC 50.000,ORI_TYP #VAR,CIRC_TYP #BASE,JERK_FAC 50.0000,GEAR_JERK 100.000,EXAX_IGN 0}

DECL E6POS XP496={X 1022,Y 549,Z -355,A 0,B -90,C 180,S 6,T 16,E1 0.0,E2 0.0,E3 0.0,E4 0.0,E5 0.0,E6 0.0}
DECL FDAT FP496={TOOL_NO 4,BASE_NO 0,IPO_FRAME #BASE,POINT2[] " "}
DECL LDAT LCPDAT496={VEL 1,ACC 50.000,APO_DIST 500.000,APO_FAC 50.0000,AXIS_VEL 50.000,AXIS_ACC 50.000,ORI_TYP #VAR,CIRC_TYP #BASE,JERK_FAC 50.0000,GEAR_JERK 100.000,EXAX_IGN 0}

DECL E6POS XP497={X 972,Y 549,Z -355,A 0,B -90,C 180,S 6,T 16,E1 0.0,E2 0.0,E3 0.0,E4 0.0,E5 0.0,E6 0.0}
DECL FDAT FP497={TOOL_NO 4,BASE_NO 0,IPO_FRAME #BASE,POINT2[] " "}
DECL LDAT LCPDAT497={VEL 1,ACC 50.000,APO_DIST 500.000,APO_FAC 50.0000,AXIS_VEL 50.000,AXIS_ACC 50.000,ORI_TYP #VAR,CIRC_TYP #BASE,JERK_FAC 50.0000,GEAR_JERK 100.000,EXAX_IGN 0}

DECL E6POS XP498={X 922,Y 549,Z -355,A 0,B -90,C 180,S 6,T 16,E1 0.0,E2 0.0,E3 0.0,E4 0.0,E5 0.0,E6 0.0}
DECL FDAT FP498={TOOL_NO 4,BASE_NO 0,IPO_FRAME #BASE,POINT2[] " "}
DECL LDAT LCPDAT498={VEL 1,ACC 50.000,APO_DIST 500.000,APO_FAC 50.0000,AXIS_VEL 50.000,AXIS_ACC 50.000,ORI_TYP #VAR,CIRC_TYP #BASE,JERK_FAC 50.0000,GEAR_JERK 100.000,EXAX_IGN 0}

DECL E6POS XP499={X 872,Y 549,Z -355,A 0,B -90,C 180,S 6,T 16,E1 0.0,E2 0.0,E3 0.0,E4 0.0,E5 0.0,E6 0.0}
DECL FDAT FP499={TOOL_NO 4,BASE_NO 0,IPO_FRAME #BASE,POINT2[] " "}
DECL LDAT LCPDAT499={VEL 1,ACC 50.000,APO_DIST 500.000,APO_FAC 50.0000,AXIS_VEL 50.000,AXIS_ACC 50.000,ORI_TYP #VAR,CIRC_TYP #BASE,JERK_FAC 50.0000,GEAR_JERK 100.000,EXAX_IGN 0}

DECL E6POS XP500={X 822,Y 549,Z -355,A 0,B -90,C 180,S 6,T 16,E1 0.0,E2 0.0,E3 0.0,E4 0.0,E5 0.0,E6 0.0}
DECL FDAT FP500={TOOL_NO 4,BASE_NO 0,IPO_FRAME #BASE,POINT2[] " "}
DECL LDAT LCPDAT500={VEL 1,ACC 50.000,APO_DIST 500.000,APO_FAC 50.0000,AXIS_VEL 50.000,AXIS_ACC 50.000,ORI_TYP #VAR,CIRC_TYP #BASE,JERK_FAC 50.0000,GEAR_JERK 100.000,EXAX_IGN 0}

DECL E6POS XP501={X 772,Y 549,Z -355,A 0,B -90,C 180,S 6,T 16,E1 0.0,E2 0.0,E3 0.0,E4 0.0,E5 0.0,E6 0.0}
DECL FDAT FP501={TOOL_NO 4,BASE_NO 0,IPO_FRAME #BASE,POINT2[] " "}
DECL LDAT LCPDAT501={VEL 1,ACC 50.000,APO_DIST 500.000,APO_FAC 50.0000,AXIS_VEL 50.000,AXIS_ACC 50.000,ORI_TYP #VAR,CIRC_TYP #BASE,JERK_FAC 50.0000,GEAR_JERK 100.000,EXAX_IGN 0}

DECL E6POS XP502={X 722,Y 549,Z -355,A 0,B -90,C 180,S 6,T 16,E1 0.0,E2 0.0,E3 0.0,E4 0.0,E5 0.0,E6 0.0}
DECL FDAT FP502={TOOL_NO 4,BASE_NO 0,IPO_FRAME #BASE,POINT2[] " "}
DECL LDAT LCPDAT502={VEL 1,ACC 50.000,APO_DIST 500.000,APO_FAC 50.0000,AXIS_VEL 50.000,AXIS_ACC 50.000,ORI_TYP #VAR,CIRC_TYP #BASE,JERK_FAC 50.0000,GEAR_JERK 100.000,EXAX_IGN 0}

DECL E6POS XP503={X 672,Y 549,Z -355,A 0,B -90,C 180,S 6,T 16,E1 0.0,E2 0.0,E3 0.0,E4 0.0,E5 0.0,E6 0.0}
DECL FDAT FP503={TOOL_NO 4,BASE_NO 0,IPO_FRAME #BASE,POINT2[] " "}
DECL LDAT LCPDAT503={VEL 1,ACC 50.000,APO_DIST 500.000,APO_FAC 50.0000,AXIS_VEL 50.000,AXIS_ACC 50.000,ORI_TYP #VAR,CIRC_TYP #BASE,JERK_FAC 50.0000,GEAR_JERK 100.000,EXAX_IGN 0}

DECL E6POS XP504={X 672,Y 549,Z -305,A 0,B -90,C 180,S 6,T 16,E1 0.0,E2 0.0,E3 0.0,E4 0.0,E5 0.0,E6 0.0}
DECL FDAT FP504={TOOL_NO 4,BASE_NO 0,IPO_FRAME #BASE,POINT2[] " "}
DECL LDAT LCPDAT504={VEL 1,ACC 50.000,APO_DIST 500.000,APO_FAC 50.0000,AXIS_VEL 50.000,AXIS_ACC 50.000,ORI_TYP #VAR,CIRC_TYP #BASE,JERK_FAC 50.0000,GEAR_JERK 100.000,EXAX_IGN 0}

DECL E6POS XP505={X 722,Y 549,Z -305,A 0,B -90,C 180,S 6,T 16,E1 0.0,E2 0.0,E3 0.0,E4 0.0,E5 0.0,E6 0.0}
DECL FDAT FP505={TOOL_NO 4,BASE_NO 0,IPO_FRAME #BASE,POINT2[] " "}
DECL LDAT LCPDAT505={VEL 1,ACC 50.000,APO_DIST 500.000,APO_FAC 50.0000,AXIS_VEL 50.000,AXIS_ACC 50.000,ORI_TYP #VAR,CIRC_TYP #BASE,JERK_FAC 50.0000,GEAR_JERK 100.000,EXAX_IGN 0}

DECL E6POS XP506={X 772,Y 549,Z -305,A 0,B -90,C 180,S 6,T 16,E1 0.0,E2 0.0,E3 0.0,E4 0.0,E5 0.0,E6 0.0}
DECL FDAT FP506={TOOL_NO 4,BASE_NO 0,IPO_FRAME #BASE,POINT2[] " "}
DECL LDAT LCPDAT506={VEL 1,ACC 50.000,APO_DIST 500.000,APO_FAC 50.0000,AXIS_VEL 50.000,AXIS_ACC 50.000,ORI_TYP #VAR,CIRC_TYP #BASE,JERK_FAC 50.0000,GEAR_JERK 100.000,EXAX_IGN 0}

DECL E6POS XP507={X 822,Y 549,Z -305,A 0,B -90,C 180,S 6,T 16,E1 0.0,E2 0.0,E3 0.0,E4 0.0,E5 0.0,E6 0.0}
DECL FDAT FP507={TOOL_NO 4,BASE_NO 0,IPO_FRAME #BASE,POINT2[] " "}
DECL LDAT LCPDAT507={VEL 1,ACC 50.000,APO_DIST 500.000,APO_FAC 50.0000,AXIS_VEL 50.000,AXIS_ACC 50.000,ORI_TYP #VAR,CIRC_TYP #BASE,JERK_FAC 50.0000,GEAR_JERK 100.000,EXAX_IGN 0}

DECL E6POS XP508={X 872,Y 549,Z -305,A 0,B -90,C 180,S 6,T 16,E1 0.0,E2 0.0,E3 0.0,E4 0.0,E5 0.0,E6 0.0}
DECL FDAT FP508={TOOL_NO 4,BASE_NO 0,IPO_FRAME #BASE,POINT2[] " "}
DECL LDAT LCPDAT508={VEL 1,ACC 50.000,APO_DIST 500.000,APO_FAC 50.0000,AXIS_VEL 50.000,AXIS_ACC 50.000,ORI_TYP #VAR,CIRC_TYP #BASE,JERK_FAC 50.0000,GEAR_JERK 100.000,EXAX_IGN 0}

DECL E6POS XP509={X 922,Y 549,Z -305,A 0,B -90,C 180,S 6,T 16,E1 0.0,E2 0.0,E3 0.0,E4 0.0,E5 0.0,E6 0.0}
DECL FDAT FP509={TOOL_NO 4,BASE_NO 0,IPO_FRAME #BASE,POINT2[] " "}
DECL LDAT LCPDAT509={VEL 1,ACC 50.000,APO_DIST 500.000,APO_FAC 50.0000,AXIS_VEL 50.000,AXIS_ACC 50.000,ORI_TYP #VAR,CIRC_TYP #BASE,JERK_FAC 50.0000,GEAR_JERK 100.000,EXAX_IGN 0}

DECL E6POS XP510={X 972,Y 549,Z -305,A 0,B -90,C 180,S 6,T 16,E1 0.0,E2 0.0,E3 0.0,E4 0.0,E5 0.0,E6 0.0}
DECL FDAT FP510={TOOL_NO 4,BASE_NO 0,IPO_FRAME #BASE,POINT2[] " "}
DECL LDAT LCPDAT510={VEL 1,ACC 50.000,APO_DIST 500.000,APO_FAC 50.0000,AXIS_VEL 50.000,AXIS_ACC 50.000,ORI_TYP #VAR,CIRC_TYP #BASE,JERK_FAC 50.0000,GEAR_JERK 100.000,EXAX_IGN 0}

DECL E6POS XP511={X 1022,Y 549,Z -305,A 0,B -90,C 180,S 6,T 16,E1 0.0,E2 0.0,E3 0.0,E4 0.0,E5 0.0,E6 0.0}
DECL FDAT FP511={TOOL_NO 4,BASE_NO 0,IPO_FRAME #BASE,POINT2[] " "}
DECL LDAT LCPDAT511={VEL 1,ACC 50.000,APO_DIST 500.000,APO_FAC 50.0000,AXIS_VEL 50.000,AXIS_ACC 50.000,ORI_TYP #VAR,CIRC_TYP #BASE,JERK_FAC 50.0000,GEAR_JERK 100.000,EXAX_IGN 0}

DECL E6POS XP512={X 1072,Y 549,Z -305,A 0,B -90,C 180,S 6,T 16,E1 0.0,E2 0.0,E3 0.0,E4 0.0,E5 0.0,E6 0.0}
DECL FDAT FP512={TOOL_NO 4,BASE_NO 0,IPO_FRAME #BASE,POINT2[] " "}
DECL LDAT LCPDAT512={VEL 1,ACC 50.000,APO_DIST 500.000,APO_FAC 50.0000,AXIS_VEL 50.000,AXIS_ACC 50.000,ORI_TYP #VAR,CIRC_TYP #BASE,JERK_FAC 50.0000,GEAR_JERK 100.000,EXAX_IGN 0}

DECL E6POS XP513={X 1122,Y 549,Z -305,A 0,B -90,C 180,S 6,T 16,E1 0.0,E2 0.0,E3 0.0,E4 0.0,E5 0.0,E6 0.0}
DECL FDAT FP513={TOOL_NO 4,BASE_NO 0,IPO_FRAME #BASE,POINT2[] " "}
DECL LDAT LCPDAT513={VEL 1,ACC 50.000,APO_DIST 500.000,APO_FAC 50.0000,AXIS_VEL 50.000,AXIS_ACC 50.000,ORI_TYP #VAR,CIRC_TYP #BASE,JERK_FAC 50.0000,GEAR_JERK 100.000,EXAX_IGN 0}

DECL E6POS XP514={X 1172,Y 549,Z -305,A 0,B -90,C 180,S 6,T 16,E1 0.0,E2 0.0,E3 0.0,E4 0.0,E5 0.0,E6 0.0}
DECL FDAT FP514={TOOL_NO 4,BASE_NO 0,IPO_FRAME #BASE,POINT2[] " "}
DECL LDAT LCPDAT514={VEL 1,ACC 50.000,APO_DIST 500.000,APO_FAC 50.0000,AXIS_VEL 50.000,AXIS_ACC 50.000,ORI_TYP #VAR,CIRC_TYP #BASE,JERK_FAC 50.0000,GEAR_JERK 100.000,EXAX_IGN 0}

DECL E6POS XP515={X 1222,Y 549,Z -305,A 0,B -90,C 180,S 6,T 16,E1 0.0,E2 0.0,E3 0.0,E4 0.0,E5 0.0,E6 0.0}
DECL FDAT FP515={TOOL_NO 4,BASE_NO 0,IPO_FRAME #BASE,POINT2[] " "}
DECL LDAT LCPDAT515={VEL 1,ACC 50.000,APO_DIST 500.000,APO_FAC 50.0000,AXIS_VEL 50.000,AXIS_ACC 50.000,ORI_TYP #VAR,CIRC_TYP #BASE,JERK_FAC 50.0000,GEAR_JERK 100.000,EXAX_IGN 0}

DECL E6POS XP516={X 1272,Y 549,Z -305,A 0,B -90,C 180,S 6,T 16,E1 0.0,E2 0.0,E3 0.0,E4 0.0,E5 0.0,E6 0.0}
DECL FDAT FP516={TOOL_NO 4,BASE_NO 0,IPO_FRAME #BASE,POINT2[] " "}
DECL LDAT LCPDAT516={VEL 1,ACC 50.000,APO_DIST 500.000,APO_FAC 50.0000,AXIS_VEL 50.000,AXIS_ACC 50.000,ORI_TYP #VAR,CIRC_TYP #BASE,JERK_FAC 50.0000,GEAR_JERK 100.000,EXAX_IGN 0}

DECL E6POS XP517={X 1272,Y 549,Z -255,A 0,B -90,C 180,S 6,T 16,E1 0.0,E2 0.0,E3 0.0,E4 0.0,E5 0.0,E6 0.0}
DECL FDAT FP517={TOOL_NO 4,BASE_NO 0,IPO_FRAME #BASE,POINT2[] " "}
DECL LDAT LCPDAT517={VEL 1,ACC 50.000,APO_DIST 500.000,APO_FAC 50.0000,AXIS_VEL 50.000,AXIS_ACC 50.000,ORI_TYP #VAR,CIRC_TYP #BASE,JERK_FAC 50.0000,GEAR_JERK 100.000,EXAX_IGN 0}

DECL E6POS XP518={X 1222,Y 549,Z -255,A 0,B -90,C 180,S 6,T 16,E1 0.0,E2 0.0,E3 0.0,E4 0.0,E5 0.0,E6 0.0}
DECL FDAT FP518={TOOL_NO 4,BASE_NO 0,IPO_FRAME #BASE,POINT2[] " "}
DECL LDAT LCPDAT518={VEL 1,ACC 50.000,APO_DIST 500.000,APO_FAC 50.0000,AXIS_VEL 50.000,AXIS_ACC 50.000,ORI_TYP #VAR,CIRC_TYP #BASE,JERK_FAC 50.0000,GEAR_JERK 100.000,EXAX_IGN 0}

DECL E6POS XP519={X 1172,Y 549,Z -255,A 0,B -90,C 180,S 6,T 16,E1 0.0,E2 0.0,E3 0.0,E4 0.0,E5 0.0,E6 0.0}
DECL FDAT FP519={TOOL_NO 4,BASE_NO 0,IPO_FRAME #BASE,POINT2[] " "}
DECL LDAT LCPDAT519={VEL 1,ACC 50.000,APO_DIST 500.000,APO_FAC 50.0000,AXIS_VEL 50.000,AXIS_ACC 50.000,ORI_TYP #VAR,CIRC_TYP #BASE,JERK_FAC 50.0000,GEAR_JERK 100.000,EXAX_IGN 0}

DECL E6POS XP520={X 1122,Y 549,Z -255,A 0,B -90,C 180,S 6,T 16,E1 0.0,E2 0.0,E3 0.0,E4 0.0,E5 0.0,E6 0.0}
DECL FDAT FP520={TOOL_NO 4,BASE_NO 0,IPO_FRAME #BASE,POINT2[] " "}
DECL LDAT LCPDAT520={VEL 1,ACC 50.000,APO_DIST 500.000,APO_FAC 50.0000,AXIS_VEL 50.000,AXIS_ACC 50.000,ORI_TYP #VAR,CIRC_TYP #BASE,JERK_FAC 50.0000,GEAR_JERK 100.000,EXAX_IGN 0}

DECL E6POS XP521={X 1072,Y 549,Z -255,A 0,B -90,C 180,S 6,T 16,E1 0.0,E2 0.0,E3 0.0,E4 0.0,E5 0.0,E6 0.0}
DECL FDAT FP521={TOOL_NO 4,BASE_NO 0,IPO_FRAME #BASE,POINT2[] " "}
DECL LDAT LCPDAT521={VEL 1,ACC 50.000,APO_DIST 500.000,APO_FAC 50.0000,AXIS_VEL 50.000,AXIS_ACC 50.000,ORI_TYP #VAR,CIRC_TYP #BASE,JERK_FAC 50.0000,GEAR_JERK 100.000,EXAX_IGN 0}

DECL E6POS XP522={X 1022,Y 549,Z -255,A 0,B -90,C 180,S 6,T 16,E1 0.0,E2 0.0,E3 0.0,E4 0.0,E5 0.0,E6 0.0}
DECL FDAT FP522={TOOL_NO 4,BASE_NO 0,IPO_FRAME #BASE,POINT2[] " "}
DECL LDAT LCPDAT522={VEL 1,ACC 50.000,APO_DIST 500.000,APO_FAC 50.0000,AXIS_VEL 50.000,AXIS_ACC 50.000,ORI_TYP #VAR,CIRC_TYP #BASE,JERK_FAC 50.0000,GEAR_JERK 100.000,EXAX_IGN 0}

DECL E6POS XP523={X 972,Y 549,Z -255,A 0,B -90,C 180,S 6,T 16,E1 0.0,E2 0.0,E3 0.0,E4 0.0,E5 0.0,E6 0.0}
DECL FDAT FP523={TOOL_NO 4,BASE_NO 0,IPO_FRAME #BASE,POINT2[] " "}
DECL LDAT LCPDAT523={VEL 1,ACC 50.000,APO_DIST 500.000,APO_FAC 50.0000,AXIS_VEL 50.000,AXIS_ACC 50.000,ORI_TYP #VAR,CIRC_TYP #BASE,JERK_FAC 50.0000,GEAR_JERK 100.000,EXAX_IGN 0}

DECL E6POS XP524={X 922,Y 549,Z -255,A 0,B -90,C 180,S 6,T 16,E1 0.0,E2 0.0,E3 0.0,E4 0.0,E5 0.0,E6 0.0}
DECL FDAT FP524={TOOL_NO 4,BASE_NO 0,IPO_FRAME #BASE,POINT2[] " "}
DECL LDAT LCPDAT524={VEL 1,ACC 50.000,APO_DIST 500.000,APO_FAC 50.0000,AXIS_VEL 50.000,AXIS_ACC 50.000,ORI_TYP #VAR,CIRC_TYP #BASE,JERK_FAC 50.0000,GEAR_JERK 100.000,EXAX_IGN 0}

DECL E6POS XP525={X 872,Y 549,Z -255,A 0,B -90,C 180,S 6,T 16,E1 0.0,E2 0.0,E3 0.0,E4 0.0,E5 0.0,E6 0.0}
DECL FDAT FP525={TOOL_NO 4,BASE_NO 0,IPO_FRAME #BASE,POINT2[] " "}
DECL LDAT LCPDAT525={VEL 1,ACC 50.000,APO_DIST 500.000,APO_FAC 50.0000,AXIS_VEL 50.000,AXIS_ACC 50.000,ORI_TYP #VAR,CIRC_TYP #BASE,JERK_FAC 50.0000,GEAR_JERK 100.000,EXAX_IGN 0}

